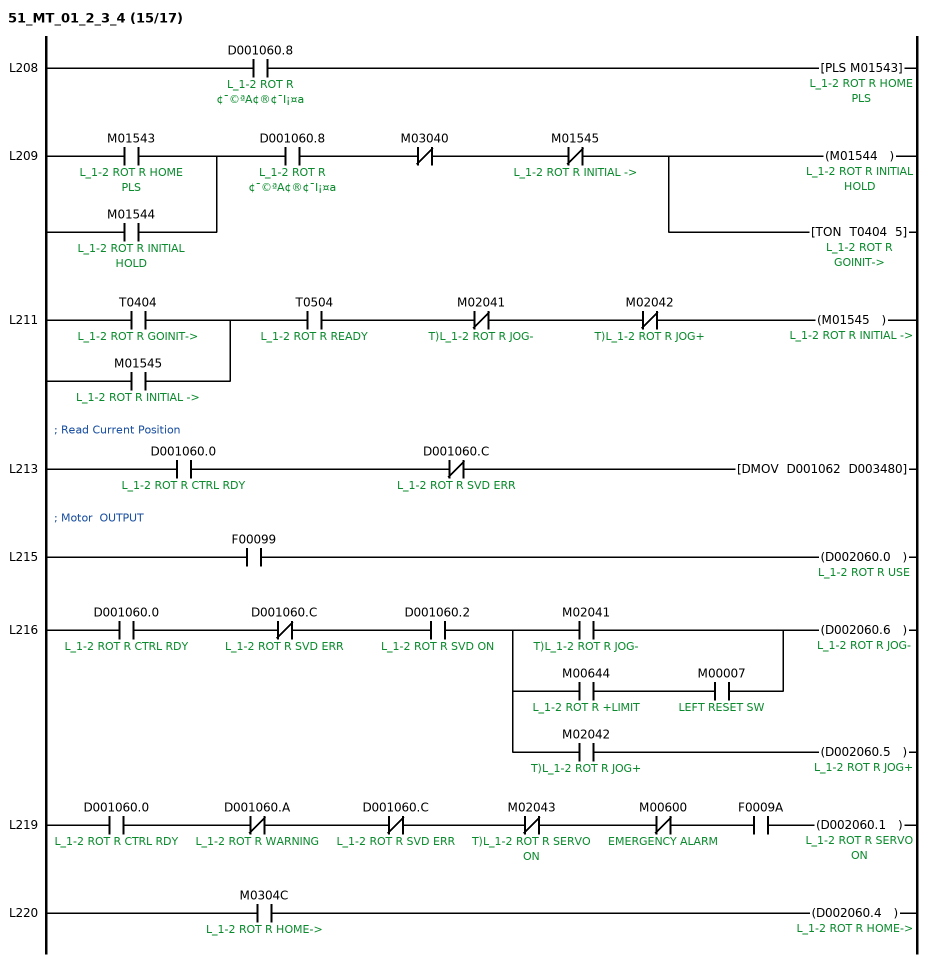
[picture p264: 51_MT_01_2_3_4 rungs L208-L220]
; L208
LOAD      D001060.8	// L_1-2 ROT R ¢¯©ªA¢®¢¯I¡¤a
OUTP      M01543	// L_1-2 ROT R HOME PLS
; L209
LOAD      M01543	// L_1-2 ROT R HOME PLS
OR        M01544	// L_1-2 ROT R INITIAL HOLD
AND       D001060.8	// L_1-2 ROT R ¢¯©ªA¢®¢¯I¡¤a
AND NOT   M03040
AND NOT   M01545	// L_1-2 ROT R INITIAL ->
OUT       M01544	// L_1-2 ROT R INITIAL HOLD
TON       T0404 5	// L_1-2 ROT R GOINIT->
; L211
LOAD      T0404	// L_1-2 ROT R GOINIT->
OR        M01545	// L_1-2 ROT R INITIAL ->
AND       T0504	// L_1-2 ROT R READY
AND NOT   M02041	// T)L_1-2 ROT R JOG-
AND NOT   M02042	// T)L_1-2 ROT R JOG+
OUT       M01545	// L_1-2 ROT R INITIAL ->
; L213
LOAD      D001060.0	// L_1-2 ROT R CTRL RDY
AND NOT   D001060.C	// L_1-2 ROT R SVD ERR
DMOV      D001062 D003480
// output comment: Read Current Position
//  Motor  OUTPUT
; L215
LOAD      F00099
OUT       D002060.0	// L_1-2 ROT R USE
; L216
LOAD      D001060.0	// L_1-2 ROT R CTRL RDY
AND NOT   D001060.C	// L_1-2 ROT R SVD ERR
AND       D001060.2	// L_1-2 ROT R SVD ON
MPUSH
LOAD      M02041	// T)L_1-2 ROT R JOG-
LOAD      M00644	// L_1-2 ROT R +LIMIT
AND       M00007	// LEFT RESET SW
OR LOAD
AND LOAD
OUT       D002060.6	// L_1-2 ROT R JOG-
MPOP
AND       M02042	// T)L_1-2 ROT R JOG+
OUT       D002060.5	// L_1-2 ROT R JOG+
; L219
LOAD      D001060.0	// L_1-2 ROT R CTRL RDY
AND NOT   D001060.A	// L_1-2 ROT R WARNING
AND NOT   D001060.C	// L_1-2 ROT R SVD ERR
AND NOT   M02043	// T)L_1-2 ROT R SERVO ON
AND NOT   M00600	// EMERGENCY ALARM
AND       F0009A
OUT       D002060.1	// L_1-2 ROT R SERVO ON
; L220
LOAD      M0304C	// L_1-2 ROT R HOME->
OUT       D002060.4	// L_1-2 ROT R HOME->

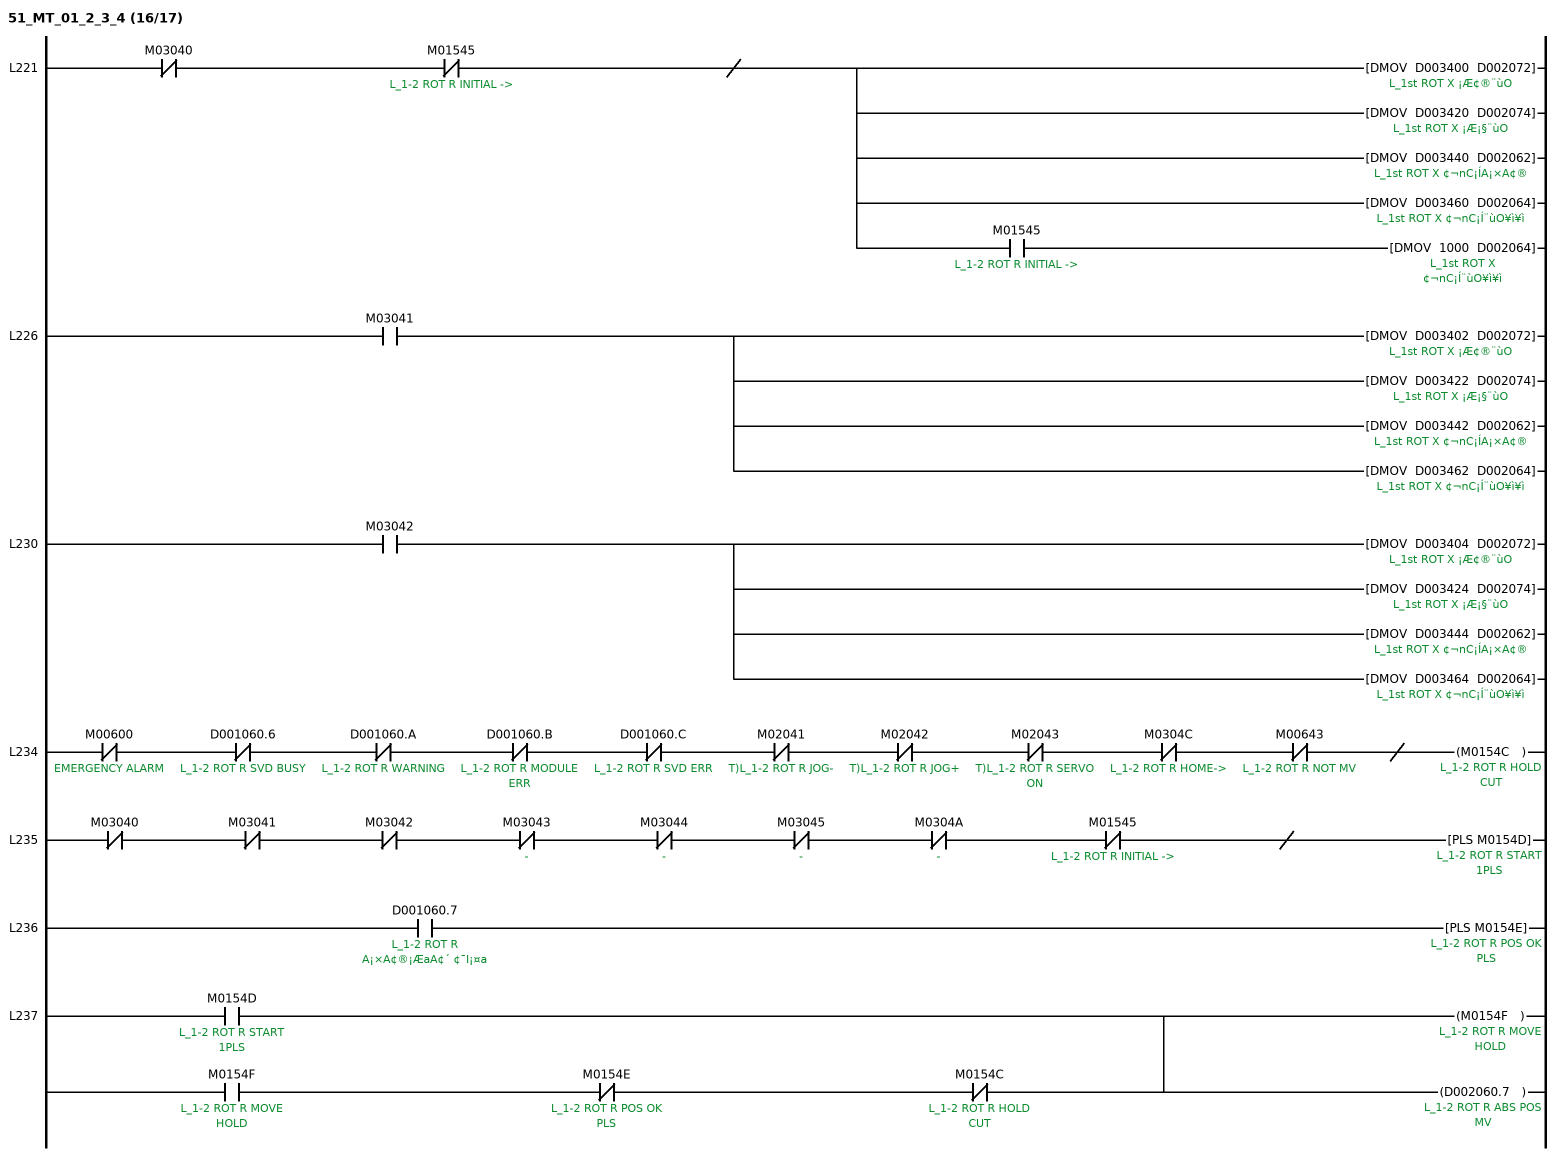
; L221
LOAD NOT  M03040
AND NOT   M01545	// L_1-2 ROT R INITIAL ->
NOT
DMOV      D003400 D002072	// L_1st ROT X ¡Æ¢®¨ùO
DMOV      D003420 D002074	// L_1st ROT X ¡Æ¡§¨ùO
DMOV      D003440 D002062	// L_1st ROT X ¢¬nC¡ÍA¡×A¢®
DMOV      D003460 D002064	// L_1st ROT X ¢¬nC¡Í¨ùO¥ì¥ì
AND       M01545	// L_1-2 ROT R INITIAL ->
DMOV      1000 D002064	// L_1st ROT X ¢¬nC¡Í¨ùO¥ì¥ì
; L226
LOAD      M03041
DMOV      D003402 D002072	// L_1st ROT X ¡Æ¢®¨ùO
DMOV      D003422 D002074	// L_1st ROT X ¡Æ¡§¨ùO
DMOV      D003442 D002062	// L_1st ROT X ¢¬nC¡ÍA¡×A¢®
DMOV      D003462 D002064	// L_1st ROT X ¢¬nC¡Í¨ùO¥ì¥ì
; L230
LOAD      M03042
DMOV      D003404 D002072	// L_1st ROT X ¡Æ¢®¨ùO
DMOV      D003424 D002074	// L_1st ROT X ¡Æ¡§¨ùO
DMOV      D003444 D002062	// L_1st ROT X ¢¬nC¡ÍA¡×A¢®
DMOV      D003464 D002064	// L_1st ROT X ¢¬nC¡Í¨ùO¥ì¥ì
; L234
LOAD NOT  M00600	// EMERGENCY ALARM
AND NOT   D001060.6	// L_1-2 ROT R SVD BUSY
AND NOT   D001060.A	// L_1-2 ROT R WARNING
AND NOT   D001060.B	// L_1-2 ROT R MODULE ERR
AND NOT   D001060.C	// L_1-2 ROT R SVD ERR
AND NOT   M02041	// T)L_1-2 ROT R JOG-
AND NOT   M02042	// T)L_1-2 ROT R JOG+
AND NOT   M02043	// T)L_1-2 ROT R SERVO ON
AND NOT   M0304C	// L_1-2 ROT R HOME->
AND NOT   M00643	// L_1-2 ROT R NOT MV
NOT
OUT       M0154C	// L_1-2 ROT R HOLD CUT
; L235
LOAD NOT  M03040
AND NOT   M03041
AND NOT   M03042
AND NOT   M03043	// -
AND NOT   M03044	// -
AND NOT   M03045	// -
AND NOT   M0304A	// -
AND NOT   M01545	// L_1-2 ROT R INITIAL ->
NOT
OUTP      M0154D	// L_1-2 ROT R START 1PLS
; L236
LOAD      D001060.7	// L_1-2 ROT R A¡×A¢®¡ÆaA¢´ ¢¯I¡¤a
OUTP      M0154E	// L_1-2 ROT R POS OK PLS
; L237
LOAD      M0154D	// L_1-2 ROT R START 1PLS
LOAD      M0154F	// L_1-2 ROT R MOVE HOLD
AND NOT   M0154E	// L_1-2 ROT R POS OK PLS
AND NOT   M0154C	// L_1-2 ROT R HOLD CUT
OR LOAD
OUT       M0154F	// L_1-2 ROT R MOVE HOLD
OUT       D002060.7	// L_1-2 ROT R ABS POS MV

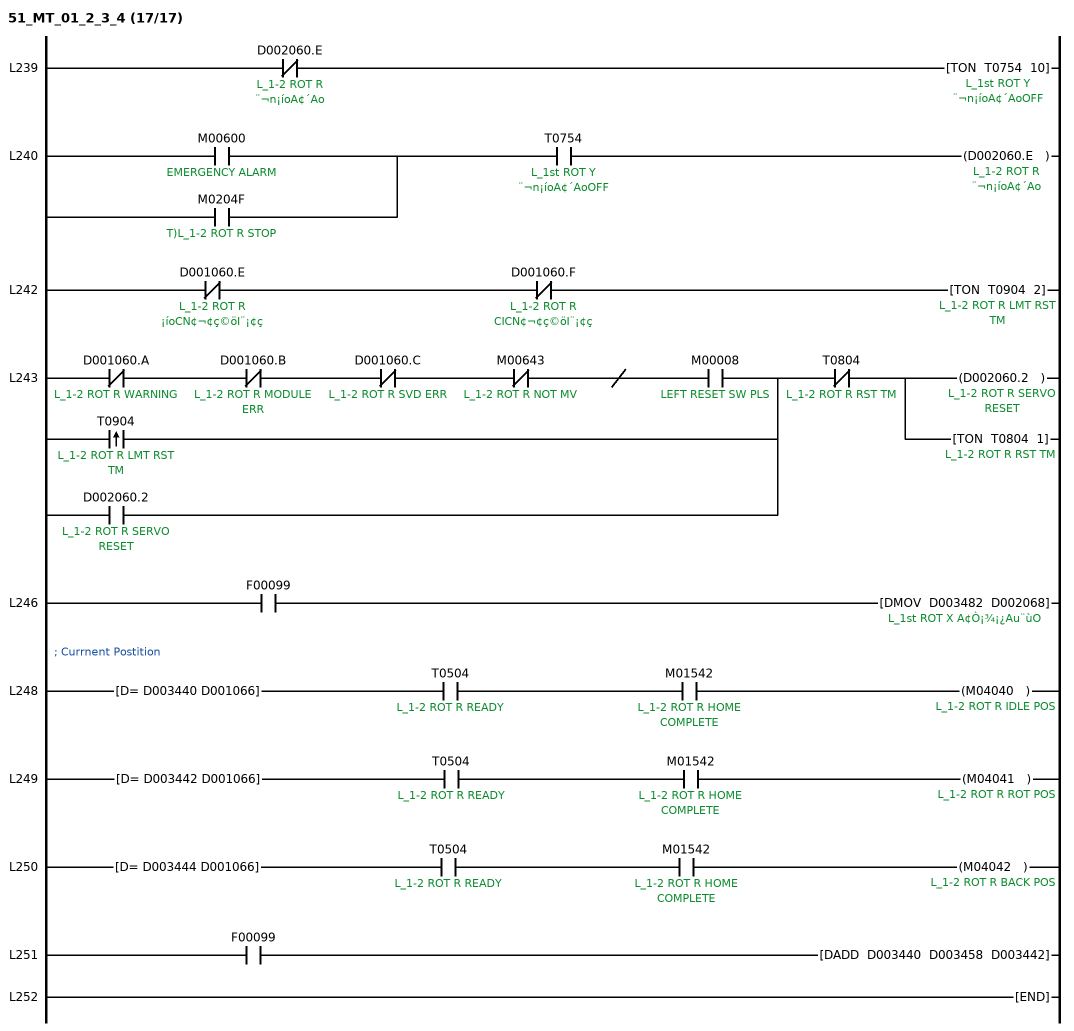
; L239
LOAD NOT  D002060.E	// L_1-2 ROT R ¨¬n¡íoA¢´Ao
TON       T0754 10	// L_1st ROT Y ¨¬n¡íoA¢´AoOFF
; L240
LOAD      M00600	// EMERGENCY ALARM
OR        M0204F	// T)L_1-2 ROT R STOP
AND       T0754	// L_1st ROT Y ¨¬n¡íoA¢´AoOFF
OUT       D002060.E	// L_1-2 ROT R ¨¬n¡íoA¢´Ao
; L242
LOAD NOT  D001060.E	// L_1-2 ROT R ¡íoCN¢¬¢ç©öI¨¡¢ç
AND NOT   D001060.F	// L_1-2 ROT R CICN¢¬¢ç©öI¨¡¢ç
TON       T0904 2	// L_1-2 ROT R LMT RST TM
; L243
LOAD NOT  D001060.A	// L_1-2 ROT R WARNING
AND NOT   D001060.B	// L_1-2 ROT R MODULE ERR
AND NOT   D001060.C	// L_1-2 ROT R SVD ERR
AND NOT   M00643	// L_1-2 ROT R NOT MV
NOT
AND       M00008	// LEFT RESET SW PLS
ORP       T0904	// L_1-2 ROT R LMT RST TM
OR        D002060.2	// L_1-2 ROT R SERVO RESET
AND NOT   T0804	// L_1-2 ROT R RST TM
OUT       D002060.2	// L_1-2 ROT R SERVO RESET
TON       T0804 1	// L_1-2 ROT R RST TM
; L246
LOAD      F00099
DMOV      D003482 D002068	// L_1st ROT X A¢Ò¡¾¡¿Au¨ùO
// Currnent Postition
; L248
LOADD=    D003440 D001066
AND       T0504	// L_1-2 ROT R READY
AND       M01542	// L_1-2 ROT R HOME COMPLETE
OUT       M04040	// L_1-2 ROT R IDLE POS
; L249
LOADD=    D003442 D001066
AND       T0504	// L_1-2 ROT R READY
AND       M01542	// L_1-2 ROT R HOME COMPLETE
OUT       M04041	// L_1-2 ROT R ROT POS
; L250
LOADD=    D003444 D001066
AND       T0504	// L_1-2 ROT R READY
AND       M01542	// L_1-2 ROT R HOME COMPLETE
OUT       M04042	// L_1-2 ROT R BACK POS
; L251
LOAD      F00099
DADD      D003440 D003458 D003442
; L252
END

PROGRAM 52_MT_05_6_7_8 (task: ¨ö¨¬A¥ì CA¡¤I¡¾¡¿¡¤¡Í)

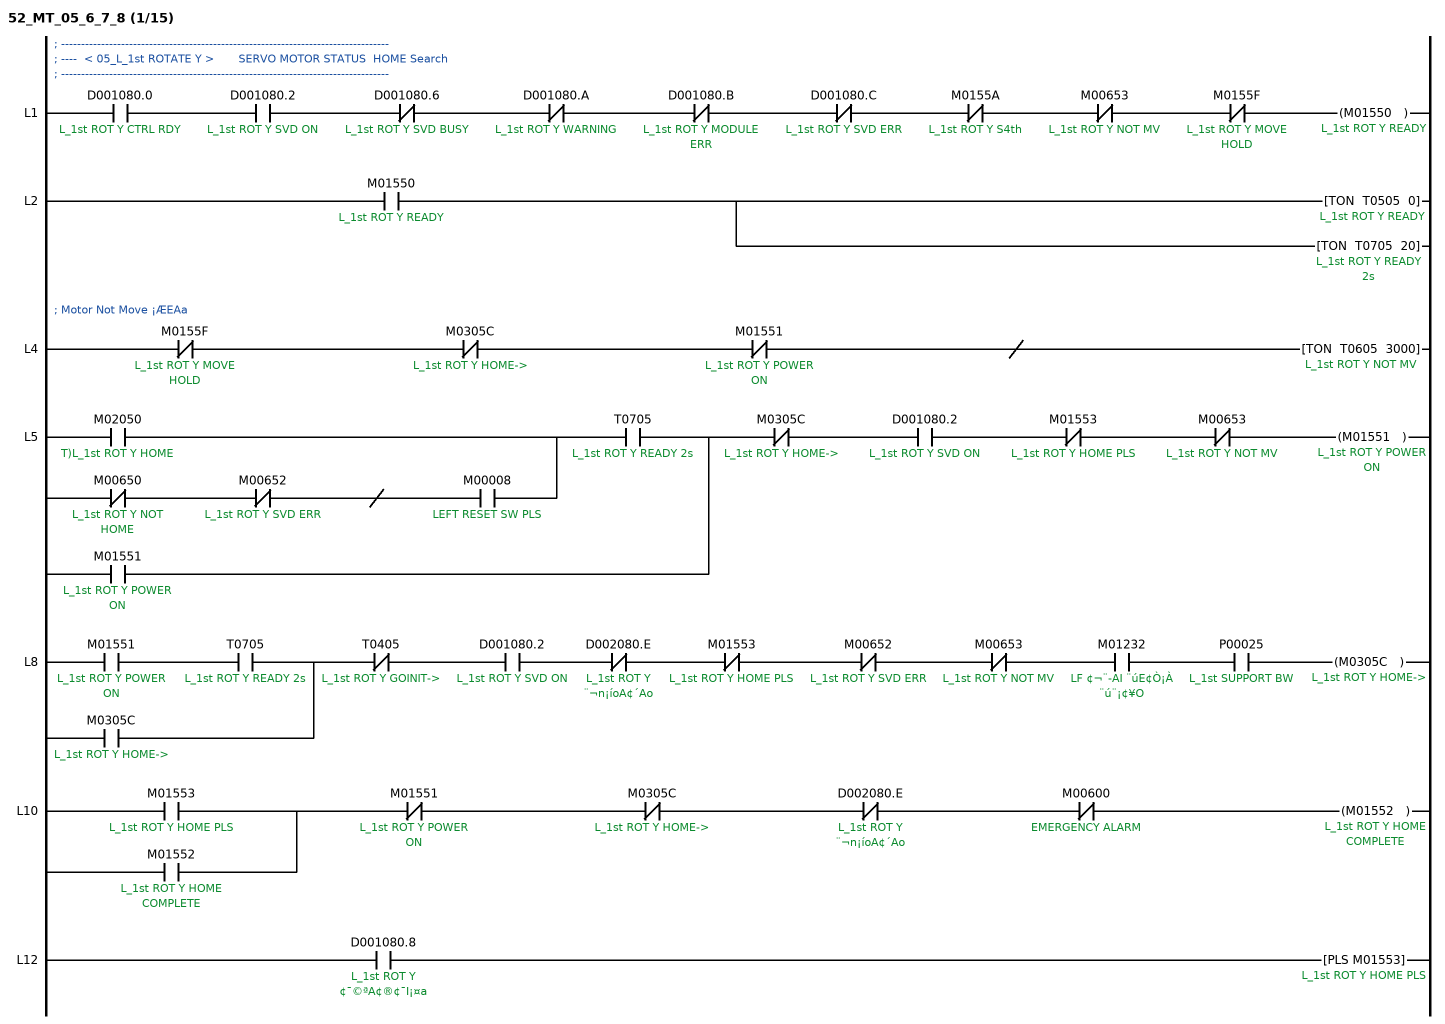
// ----------------------------------------------------------------------------------
// 
// ----  < 05_L_1st ROTATE Y >       SERVO MOTOR STATUS  HOME Search
// 
// ----------------------------------------------------------------------------------
; L1
LOAD      D001080.0	// L_1st ROT Y CTRL RDY
AND       D001080.2	// L_1st ROT Y SVD ON
AND NOT   D001080.6	// L_1st ROT Y SVD BUSY
AND NOT   D001080.A	// L_1st ROT Y WARNING
AND NOT   D001080.B	// L_1st ROT Y MODULE ERR
AND NOT   D001080.C	// L_1st ROT Y SVD ERR
AND NOT   M0155A	// L_1st ROT Y S4th
AND NOT   M00653	// L_1st ROT Y NOT MV
AND NOT   M0155F	// L_1st ROT Y MOVE HOLD
OUT       M01550	// L_1st ROT Y READY
; L2
LOAD      M01550	// L_1st ROT Y READY
TON       T0505 0	// L_1st ROT Y READY
TON       T0705 20	// L_1st ROT Y READY 2s
; L4
LOAD NOT  M0155F	// L_1st ROT Y MOVE HOLD
AND NOT   M0305C	// L_1st ROT Y HOME->
AND NOT   M01551	// L_1st ROT Y POWER ON
NOT
TON       T0605 3000	// L_1st ROT Y NOT MV
// output comment: Motor Not Move ¡ÆEAa
; L5
LOAD      M02050	// T)L_1st ROT Y HOME
LOAD NOT  M00650	// L_1st ROT Y NOT HOME
AND NOT   M00652	// L_1st ROT Y SVD ERR
NOT
AND       M00008	// LEFT RESET SW PLS
OR LOAD
AND       T0705	// L_1st ROT Y READY 2s
OR        M01551	// L_1st ROT Y POWER ON
AND NOT   M0305C	// L_1st ROT Y HOME->
AND       D001080.2	// L_1st ROT Y SVD ON
AND NOT   M01553	// L_1st ROT Y HOME PLS
AND NOT   M00653	// L_1st ROT Y NOT MV
OUT       M01551	// L_1st ROT Y POWER ON
; L8
LOAD      M01551	// L_1st ROT Y POWER ON
AND       T0705	// L_1st ROT Y READY 2s
OR        M0305C	// L_1st ROT Y HOME->
AND NOT   T0405	// L_1st ROT Y GOINIT->
AND       D001080.2	// L_1st ROT Y SVD ON
AND NOT   D002080.E	// L_1st ROT Y ¨¬n¡íoA¢´Ao
AND NOT   M01553	// L_1st ROT Y HOME PLS
AND NOT   M00652	// L_1st ROT Y SVD ERR
AND NOT   M00653	// L_1st ROT Y NOT MV
AND       M01232	// LF ¢¬¨­AI ¨úE¢Ò¡À ¨ú¨¡¢¥O
AND       P00025	// L_1st SUPPORT BW
OUT       M0305C	// L_1st ROT Y HOME->
; L10
LOAD      M01553	// L_1st ROT Y HOME PLS
OR        M01552	// L_1st ROT Y HOME COMPLETE
AND NOT   M01551	// L_1st ROT Y POWER ON
AND NOT   M0305C	// L_1st ROT Y HOME->
AND NOT   D002080.E	// L_1st ROT Y ¨¬n¡íoA¢´Ao
AND NOT   M00600	// EMERGENCY ALARM
OUT       M01552	// L_1st ROT Y HOME COMPLETE
; L12
LOAD      D001080.8	// L_1st ROT Y ¢¯©ªA¢®¢¯I¡¤a
OUTP      M01553	// L_1st ROT Y HOME PLS

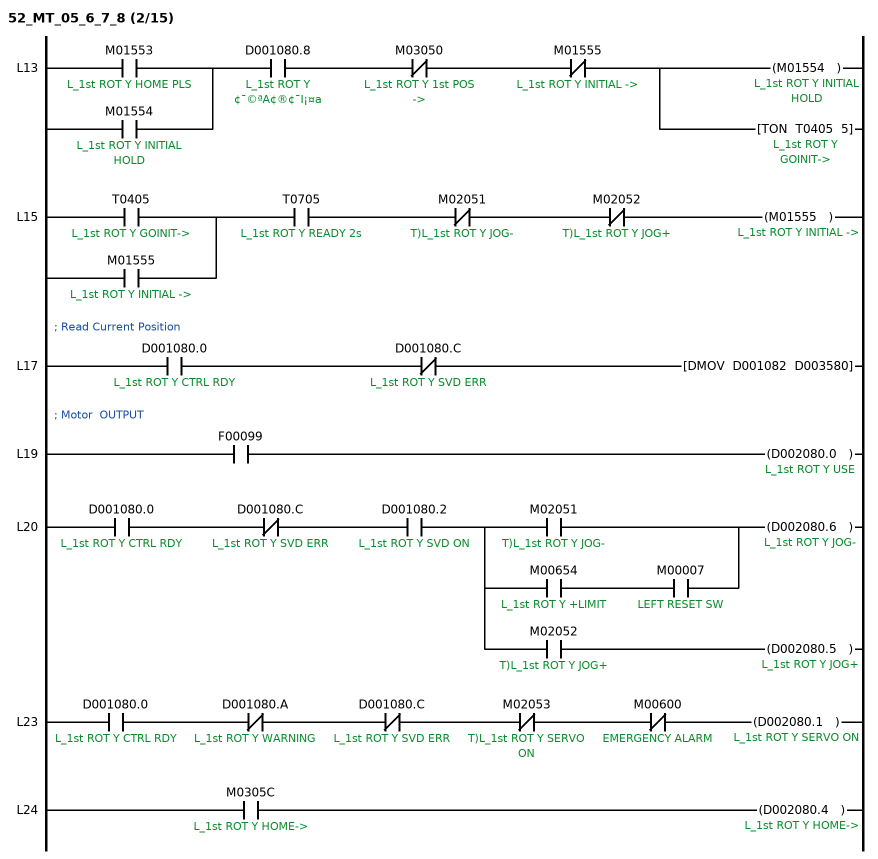
; L13
LOAD      M01553	// L_1st ROT Y HOME PLS
OR        M01554	// L_1st ROT Y INITIAL HOLD
AND       D001080.8	// L_1st ROT Y ¢¯©ªA¢®¢¯I¡¤a
AND NOT   M03050	// L_1st ROT Y 1st POS ->
AND NOT   M01555	// L_1st ROT Y INITIAL ->
OUT       M01554	// L_1st ROT Y INITIAL HOLD
TON       T0405 5	// L_1st ROT Y GOINIT->
; L15
LOAD      T0405	// L_1st ROT Y GOINIT->
OR        M01555	// L_1st ROT Y INITIAL ->
AND       T0705	// L_1st ROT Y READY 2s
AND NOT   M02051	// T)L_1st ROT Y JOG-
AND NOT   M02052	// T)L_1st ROT Y JOG+
OUT       M01555	// L_1st ROT Y INITIAL ->
; L17
LOAD      D001080.0	// L_1st ROT Y CTRL RDY
AND NOT   D001080.C	// L_1st ROT Y SVD ERR
DMOV      D001082 D003580
// output comment: Read Current Position
//  Motor  OUTPUT
; L19
LOAD      F00099
OUT       D002080.0	// L_1st ROT Y USE
; L20
LOAD      D001080.0	// L_1st ROT Y CTRL RDY
AND NOT   D001080.C	// L_1st ROT Y SVD ERR
AND       D001080.2	// L_1st ROT Y SVD ON
MPUSH
LOAD      M02051	// T)L_1st ROT Y JOG-
LOAD      M00654	// L_1st ROT Y +LIMIT
AND       M00007	// LEFT RESET SW
OR LOAD
AND LOAD
OUT       D002080.6	// L_1st ROT Y JOG-
MPOP
AND       M02052	// T)L_1st ROT Y JOG+
OUT       D002080.5	// L_1st ROT Y JOG+
; L23
LOAD      D001080.0	// L_1st ROT Y CTRL RDY
AND NOT   D001080.A	// L_1st ROT Y WARNING
AND NOT   D001080.C	// L_1st ROT Y SVD ERR
AND NOT   M02053	// T)L_1st ROT Y SERVO ON
AND NOT   M00600	// EMERGENCY ALARM
OUT       D002080.1	// L_1st ROT Y SERVO ON
; L24
LOAD      M0305C	// L_1st ROT Y HOME->
OUT       D002080.4	// L_1st ROT Y HOME->

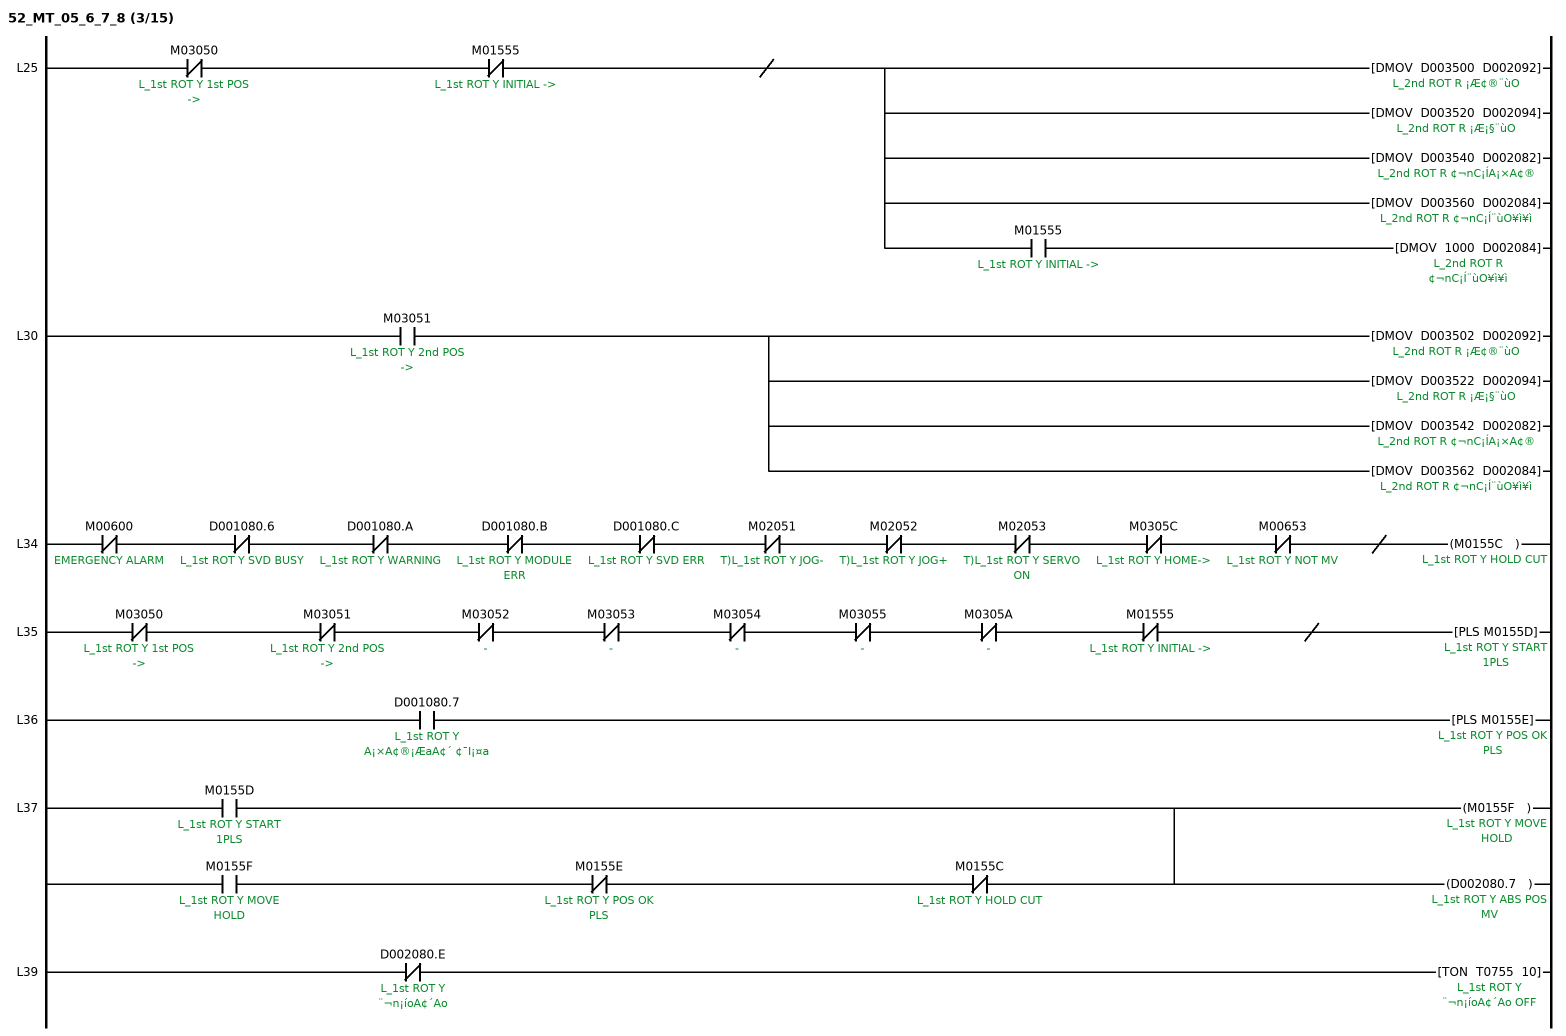
; L25
LOAD NOT  M03050	// L_1st ROT Y 1st POS ->
AND NOT   M01555	// L_1st ROT Y INITIAL ->
NOT
DMOV      D003500 D002092	// L_2nd ROT R ¡Æ¢®¨ùO
DMOV      D003520 D002094	// L_2nd ROT R ¡Æ¡§¨ùO
DMOV      D003540 D002082	// L_2nd ROT R ¢¬nC¡ÍA¡×A¢®
DMOV      D003560 D002084	// L_2nd ROT R ¢¬nC¡Í¨ùO¥ì¥ì
AND       M01555	// L_1st ROT Y INITIAL ->
DMOV      1000 D002084	// L_2nd ROT R ¢¬nC¡Í¨ùO¥ì¥ì
; L30
LOAD      M03051	// L_1st ROT Y 2nd POS ->
DMOV      D003502 D002092	// L_2nd ROT R ¡Æ¢®¨ùO
DMOV      D003522 D002094	// L_2nd ROT R ¡Æ¡§¨ùO
DMOV      D003542 D002082	// L_2nd ROT R ¢¬nC¡ÍA¡×A¢®
DMOV      D003562 D002084	// L_2nd ROT R ¢¬nC¡Í¨ùO¥ì¥ì
; L34
LOAD NOT  M00600	// EMERGENCY ALARM
AND NOT   D001080.6	// L_1st ROT Y SVD BUSY
AND NOT   D001080.A	// L_1st ROT Y WARNING
AND NOT   D001080.B	// L_1st ROT Y MODULE ERR
AND NOT   D001080.C	// L_1st ROT Y SVD ERR
AND NOT   M02051	// T)L_1st ROT Y JOG-
AND NOT   M02052	// T)L_1st ROT Y JOG+
AND NOT   M02053	// T)L_1st ROT Y SERVO ON
AND NOT   M0305C	// L_1st ROT Y HOME->
AND NOT   M00653	// L_1st ROT Y NOT MV
NOT
OUT       M0155C	// L_1st ROT Y HOLD CUT
; L35
LOAD NOT  M03050	// L_1st ROT Y 1st POS ->
AND NOT   M03051	// L_1st ROT Y 2nd POS ->
AND NOT   M03052	// -
AND NOT   M03053	// -
AND NOT   M03054	// -
AND NOT   M03055	// -
AND NOT   M0305A	// -
AND NOT   M01555	// L_1st ROT Y INITIAL ->
NOT
OUTP      M0155D	// L_1st ROT Y START 1PLS
; L36
LOAD      D001080.7	// L_1st ROT Y A¡×A¢®¡ÆaA¢´ ¢¯I¡¤a
OUTP      M0155E	// L_1st ROT Y POS OK PLS
; L37
LOAD      M0155D	// L_1st ROT Y START 1PLS
LOAD      M0155F	// L_1st ROT Y MOVE HOLD
AND NOT   M0155E	// L_1st ROT Y POS OK PLS
AND NOT   M0155C	// L_1st ROT Y HOLD CUT
OR LOAD
OUT       M0155F	// L_1st ROT Y MOVE HOLD
OUT       D002080.7	// L_1st ROT Y ABS POS MV
; L39
LOAD NOT  D002080.E	// L_1st ROT Y ¨¬n¡íoA¢´Ao
TON       T0755 10	// L_1st ROT Y ¨¬n¡íoA¢´Ao OFF

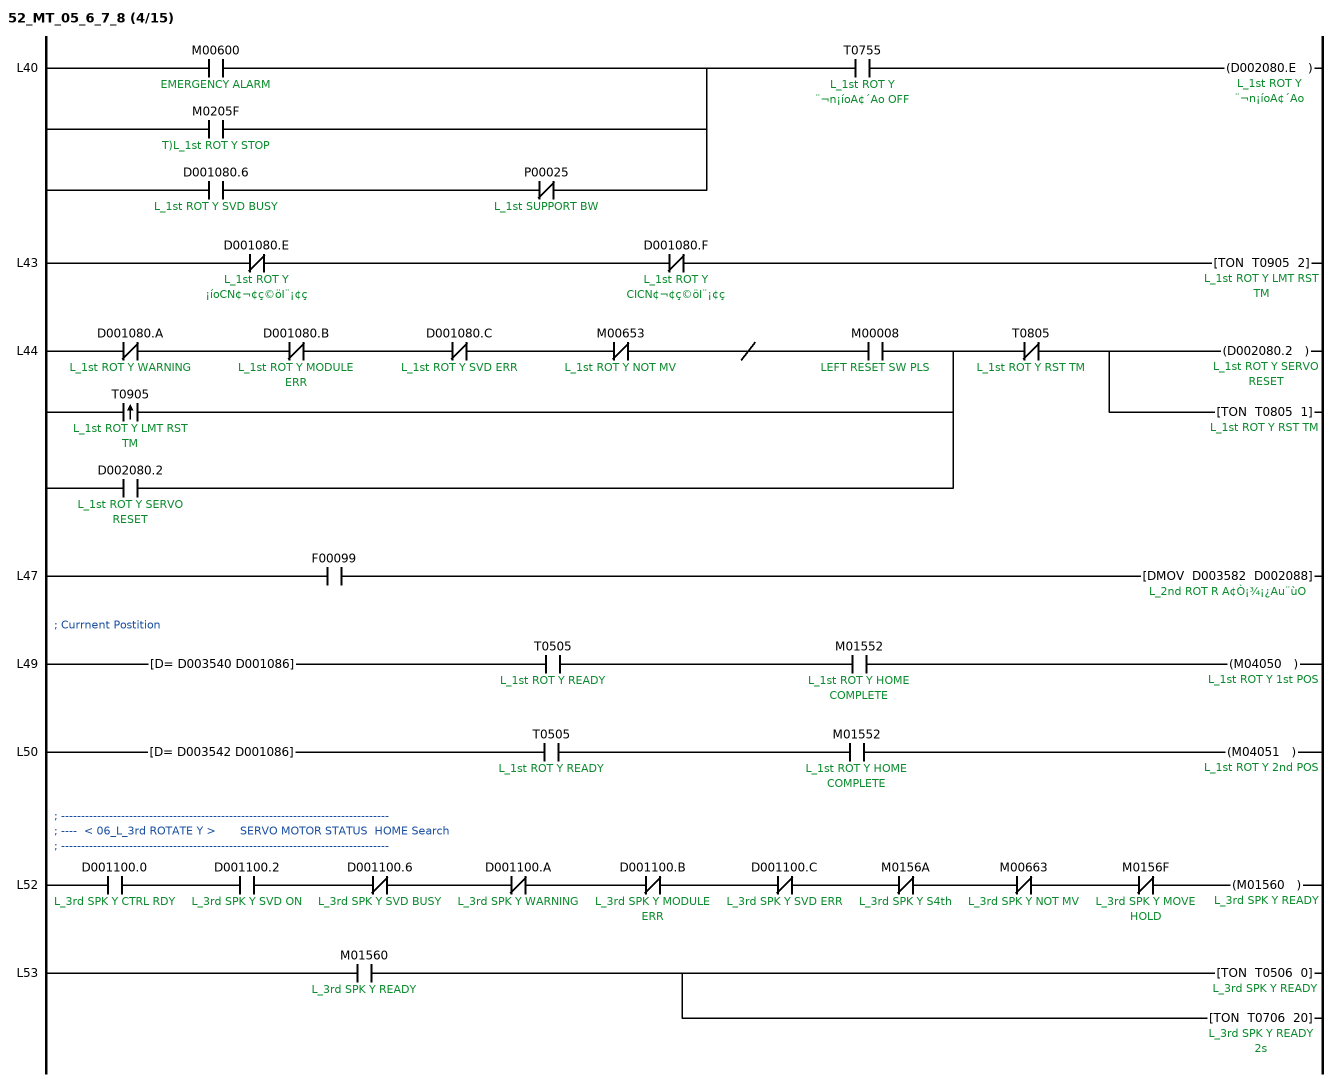
; L40
LOAD      M00600	// EMERGENCY ALARM
OR        M0205F	// T)L_1st ROT Y STOP
LOAD      D001080.6	// L_1st ROT Y SVD BUSY
AND NOT   P00025	// L_1st SUPPORT BW
OR LOAD
AND       T0755	// L_1st ROT Y ¨¬n¡íoA¢´Ao OFF
OUT       D002080.E	// L_1st ROT Y ¨¬n¡íoA¢´Ao
; L43
LOAD NOT  D001080.E	// L_1st ROT Y ¡íoCN¢¬¢ç©öI¨¡¢ç
AND NOT   D001080.F	// L_1st ROT Y CICN¢¬¢ç©öI¨¡¢ç
TON       T0905 2	// L_1st ROT Y LMT RST TM
; L44
LOAD NOT  D001080.A	// L_1st ROT Y WARNING
AND NOT   D001080.B	// L_1st ROT Y MODULE ERR
AND NOT   D001080.C	// L_1st ROT Y SVD ERR
AND NOT   M00653	// L_1st ROT Y NOT MV
NOT
AND       M00008	// LEFT RESET SW PLS
ORP       T0905	// L_1st ROT Y LMT RST TM
OR        D002080.2	// L_1st ROT Y SERVO RESET
AND NOT   T0805	// L_1st ROT Y RST TM
OUT       D002080.2	// L_1st ROT Y SERVO RESET
TON       T0805 1	// L_1st ROT Y RST TM
; L47
LOAD      F00099
DMOV      D003582 D002088	// L_2nd ROT R A¢Ò¡¾¡¿Au¨ùO
// Currnent Postition
; L49
LOADD=    D003540 D001086
AND       T0505	// L_1st ROT Y READY
AND       M01552	// L_1st ROT Y HOME COMPLETE
OUT       M04050	// L_1st ROT Y 1st POS
; L50
LOADD=    D003542 D001086
AND       T0505	// L_1st ROT Y READY
AND       M01552	// L_1st ROT Y HOME COMPLETE
OUT       M04051	// L_1st ROT Y 2nd POS
// ----------------------------------------------------------------------------------
// 
// ----  < 06_L_3rd ROTATE Y >       SERVO MOTOR STATUS  HOME Search
// 
// ----------------------------------------------------------------------------------
; L52
LOAD      D001100.0	// L_3rd SPK Y CTRL RDY
AND       D001100.2	// L_3rd SPK Y SVD ON
AND NOT   D001100.6	// L_3rd SPK Y SVD BUSY
AND NOT   D001100.A	// L_3rd SPK Y WARNING
AND NOT   D001100.B	// L_3rd SPK Y MODULE ERR
AND NOT   D001100.C	// L_3rd SPK Y SVD ERR
AND NOT   M0156A	// L_3rd SPK Y S4th
AND NOT   M00663	// L_3rd SPK Y NOT MV
AND NOT   M0156F	// L_3rd SPK Y MOVE HOLD
OUT       M01560	// L_3rd SPK Y READY
; L53
LOAD      M01560	// L_3rd SPK Y READY
TON       T0506 0	// L_3rd SPK Y READY
TON       T0706 20	// L_3rd SPK Y READY 2s

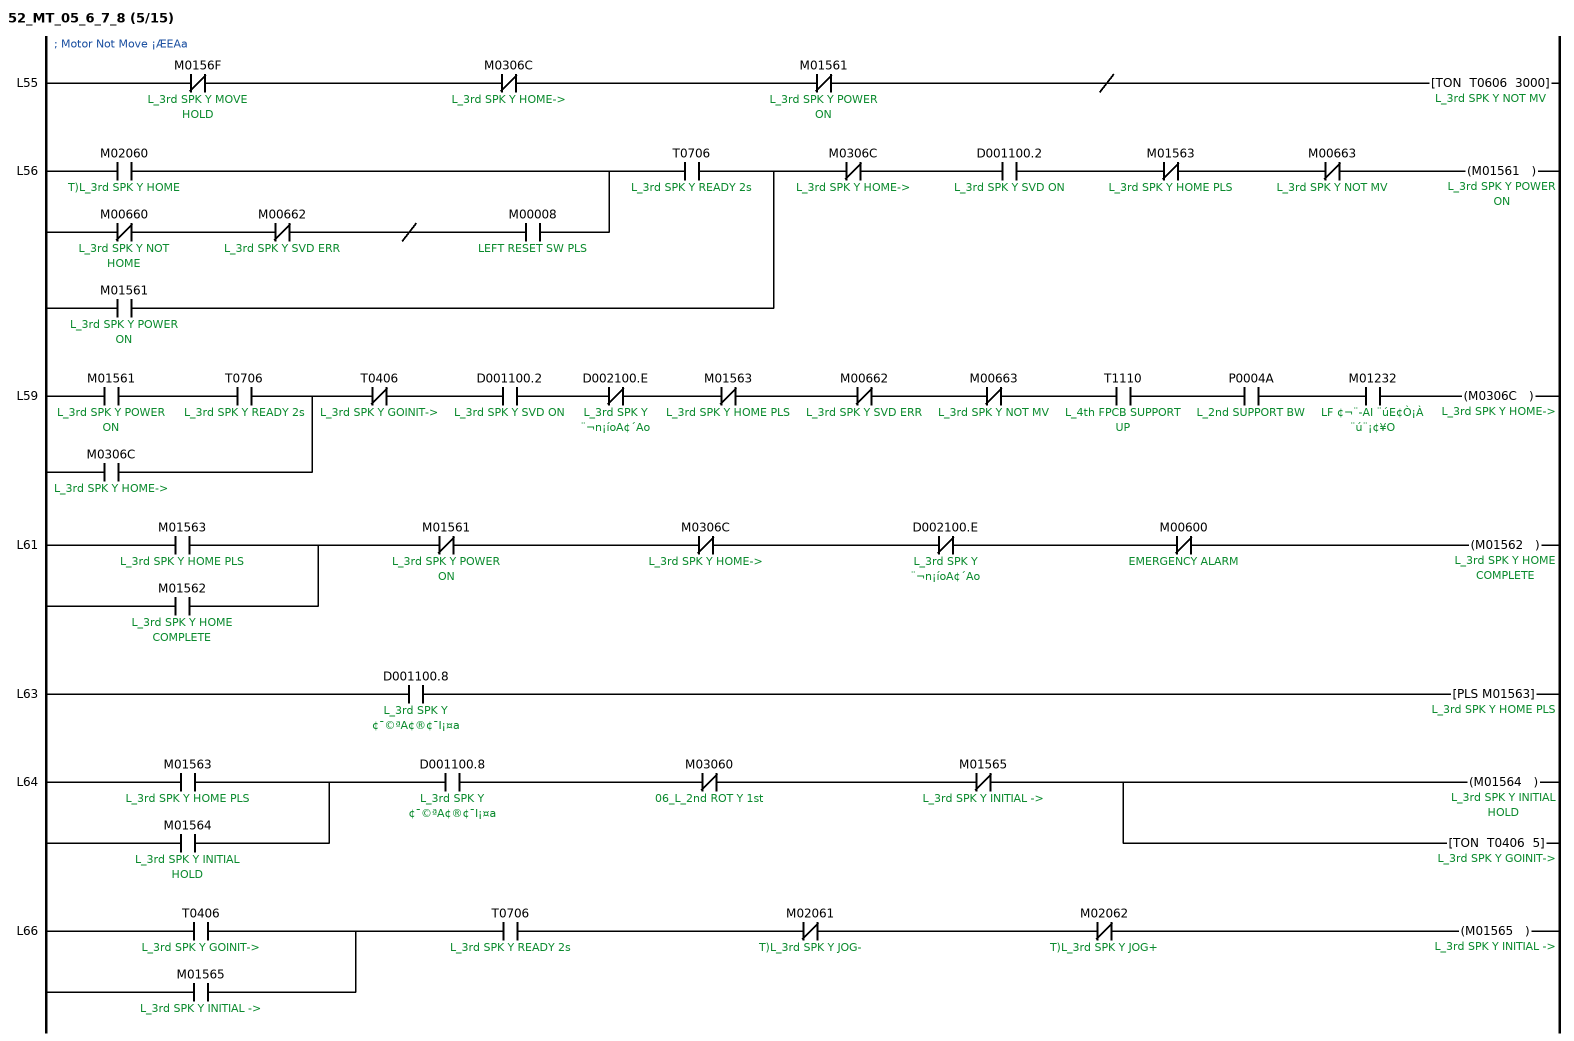
; L55
LOAD NOT  M0156F	// L_3rd SPK Y MOVE HOLD
AND NOT   M0306C	// L_3rd SPK Y HOME->
AND NOT   M01561	// L_3rd SPK Y POWER ON
NOT
TON       T0606 3000	// L_3rd SPK Y NOT MV
// output comment: Motor Not Move ¡ÆEAa
; L56
LOAD      M02060	// T)L_3rd SPK Y HOME
LOAD NOT  M00660	// L_3rd SPK Y NOT HOME
AND NOT   M00662	// L_3rd SPK Y SVD ERR
NOT
AND       M00008	// LEFT RESET SW PLS
OR LOAD
AND       T0706	// L_3rd SPK Y READY 2s
OR        M01561	// L_3rd SPK Y POWER ON
AND NOT   M0306C	// L_3rd SPK Y HOME->
AND       D001100.2	// L_3rd SPK Y SVD ON
AND NOT   M01563	// L_3rd SPK Y HOME PLS
AND NOT   M00663	// L_3rd SPK Y NOT MV
OUT       M01561	// L_3rd SPK Y POWER ON
; L59
LOAD      M01561	// L_3rd SPK Y POWER ON
AND       T0706	// L_3rd SPK Y READY 2s
OR        M0306C	// L_3rd SPK Y HOME->
AND NOT   T0406	// L_3rd SPK Y GOINIT->
AND       D001100.2	// L_3rd SPK Y SVD ON
AND NOT   D002100.E	// L_3rd SPK Y ¨¬n¡íoA¢´Ao
AND NOT   M01563	// L_3rd SPK Y HOME PLS
AND NOT   M00662	// L_3rd SPK Y SVD ERR
AND NOT   M00663	// L_3rd SPK Y NOT MV
AND       T1110	// L_4th FPCB SUPPORT UP
AND       P0004A	// L_2nd SUPPORT BW
AND       M01232	// LF ¢¬¨­AI ¨úE¢Ò¡À ¨ú¨¡¢¥O
OUT       M0306C	// L_3rd SPK Y HOME->
; L61
LOAD      M01563	// L_3rd SPK Y HOME PLS
OR        M01562	// L_3rd SPK Y HOME COMPLETE
AND NOT   M01561	// L_3rd SPK Y POWER ON
AND NOT   M0306C	// L_3rd SPK Y HOME->
AND NOT   D002100.E	// L_3rd SPK Y ¨¬n¡íoA¢´Ao
AND NOT   M00600	// EMERGENCY ALARM
OUT       M01562	// L_3rd SPK Y HOME COMPLETE
; L63
LOAD      D001100.8	// L_3rd SPK Y ¢¯©ªA¢®¢¯I¡¤a
OUTP      M01563	// L_3rd SPK Y HOME PLS
; L64
LOAD      M01563	// L_3rd SPK Y HOME PLS
OR        M01564	// L_3rd SPK Y INITIAL HOLD
AND       D001100.8	// L_3rd SPK Y ¢¯©ªA¢®¢¯I¡¤a
AND NOT   M03060	// 06_L_2nd ROT Y 1st
AND NOT   M01565	// L_3rd SPK Y INITIAL ->
OUT       M01564	// L_3rd SPK Y INITIAL HOLD
TON       T0406 5	// L_3rd SPK Y GOINIT->
; L66
LOAD      T0406	// L_3rd SPK Y GOINIT->
OR        M01565	// L_3rd SPK Y INITIAL ->
AND       T0706	// L_3rd SPK Y READY 2s
AND NOT   M02061	// T)L_3rd SPK Y JOG-
AND NOT   M02062	// T)L_3rd SPK Y JOG+
OUT       M01565	// L_3rd SPK Y INITIAL ->

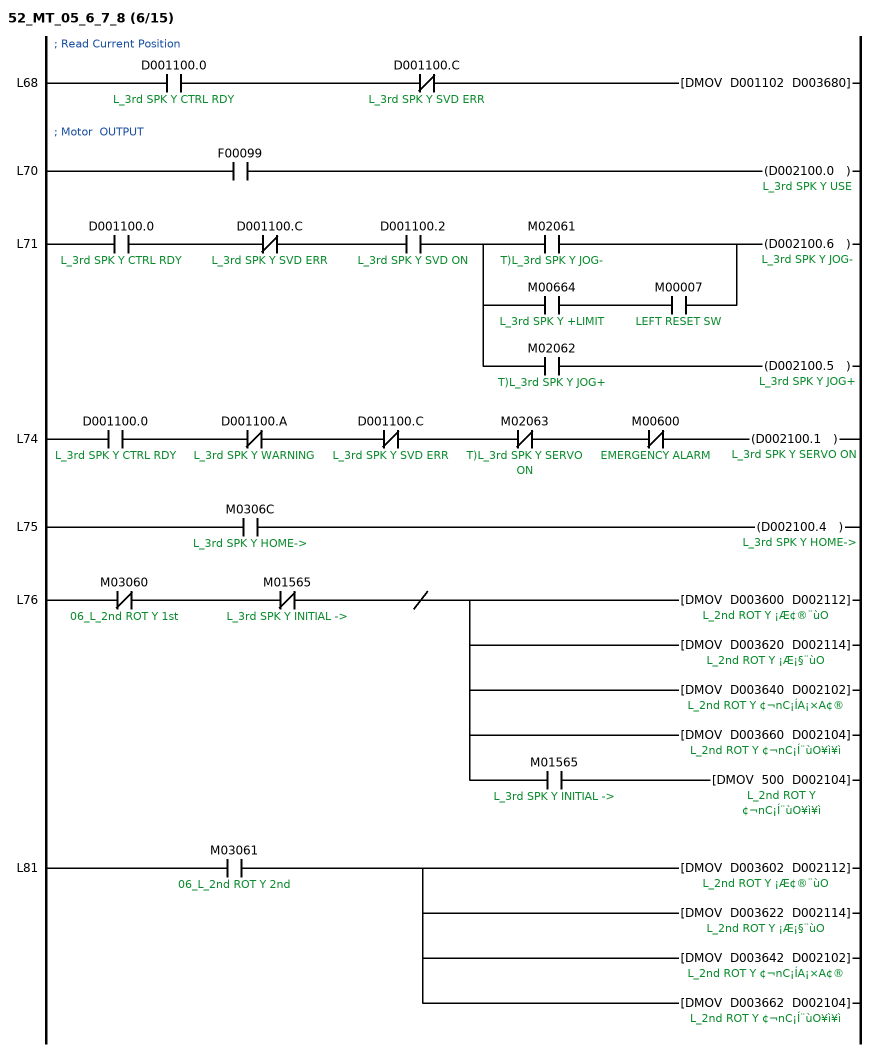
; L68
LOAD      D001100.0	// L_3rd SPK Y CTRL RDY
AND NOT   D001100.C	// L_3rd SPK Y SVD ERR
DMOV      D001102 D003680
// output comment: Read Current Position
//  Motor  OUTPUT
; L70
LOAD      F00099
OUT       D002100.0	// L_3rd SPK Y USE
; L71
LOAD      D001100.0	// L_3rd SPK Y CTRL RDY
AND NOT   D001100.C	// L_3rd SPK Y SVD ERR
AND       D001100.2	// L_3rd SPK Y SVD ON
MPUSH
LOAD      M02061	// T)L_3rd SPK Y JOG-
LOAD      M00664	// L_3rd SPK Y +LIMIT
AND       M00007	// LEFT RESET SW
OR LOAD
AND LOAD
OUT       D002100.6	// L_3rd SPK Y JOG-
MPOP
AND       M02062	// T)L_3rd SPK Y JOG+
OUT       D002100.5	// L_3rd SPK Y JOG+
; L74
LOAD      D001100.0	// L_3rd SPK Y CTRL RDY
AND NOT   D001100.A	// L_3rd SPK Y WARNING
AND NOT   D001100.C	// L_3rd SPK Y SVD ERR
AND NOT   M02063	// T)L_3rd SPK Y SERVO ON
AND NOT   M00600	// EMERGENCY ALARM
OUT       D002100.1	// L_3rd SPK Y SERVO ON
; L75
LOAD      M0306C	// L_3rd SPK Y HOME->
OUT       D002100.4	// L_3rd SPK Y HOME->
; L76
LOAD NOT  M03060	// 06_L_2nd ROT Y 1st
AND NOT   M01565	// L_3rd SPK Y INITIAL ->
NOT
DMOV      D003600 D002112	// L_2nd ROT Y ¡Æ¢®¨ùO
DMOV      D003620 D002114	// L_2nd ROT Y ¡Æ¡§¨ùO
DMOV      D003640 D002102	// L_2nd ROT Y ¢¬nC¡ÍA¡×A¢®
DMOV      D003660 D002104	// L_2nd ROT Y ¢¬nC¡Í¨ùO¥ì¥ì
AND       M01565	// L_3rd SPK Y INITIAL ->
DMOV      500 D002104	// L_2nd ROT Y ¢¬nC¡Í¨ùO¥ì¥ì
; L81
LOAD      M03061	// 06_L_2nd ROT Y 2nd
DMOV      D003602 D002112	// L_2nd ROT Y ¡Æ¢®¨ùO
DMOV      D003622 D002114	// L_2nd ROT Y ¡Æ¡§¨ùO
DMOV      D003642 D002102	// L_2nd ROT Y ¢¬nC¡ÍA¡×A¢®
DMOV      D003662 D002104	// L_2nd ROT Y ¢¬nC¡Í¨ùO¥ì¥ì

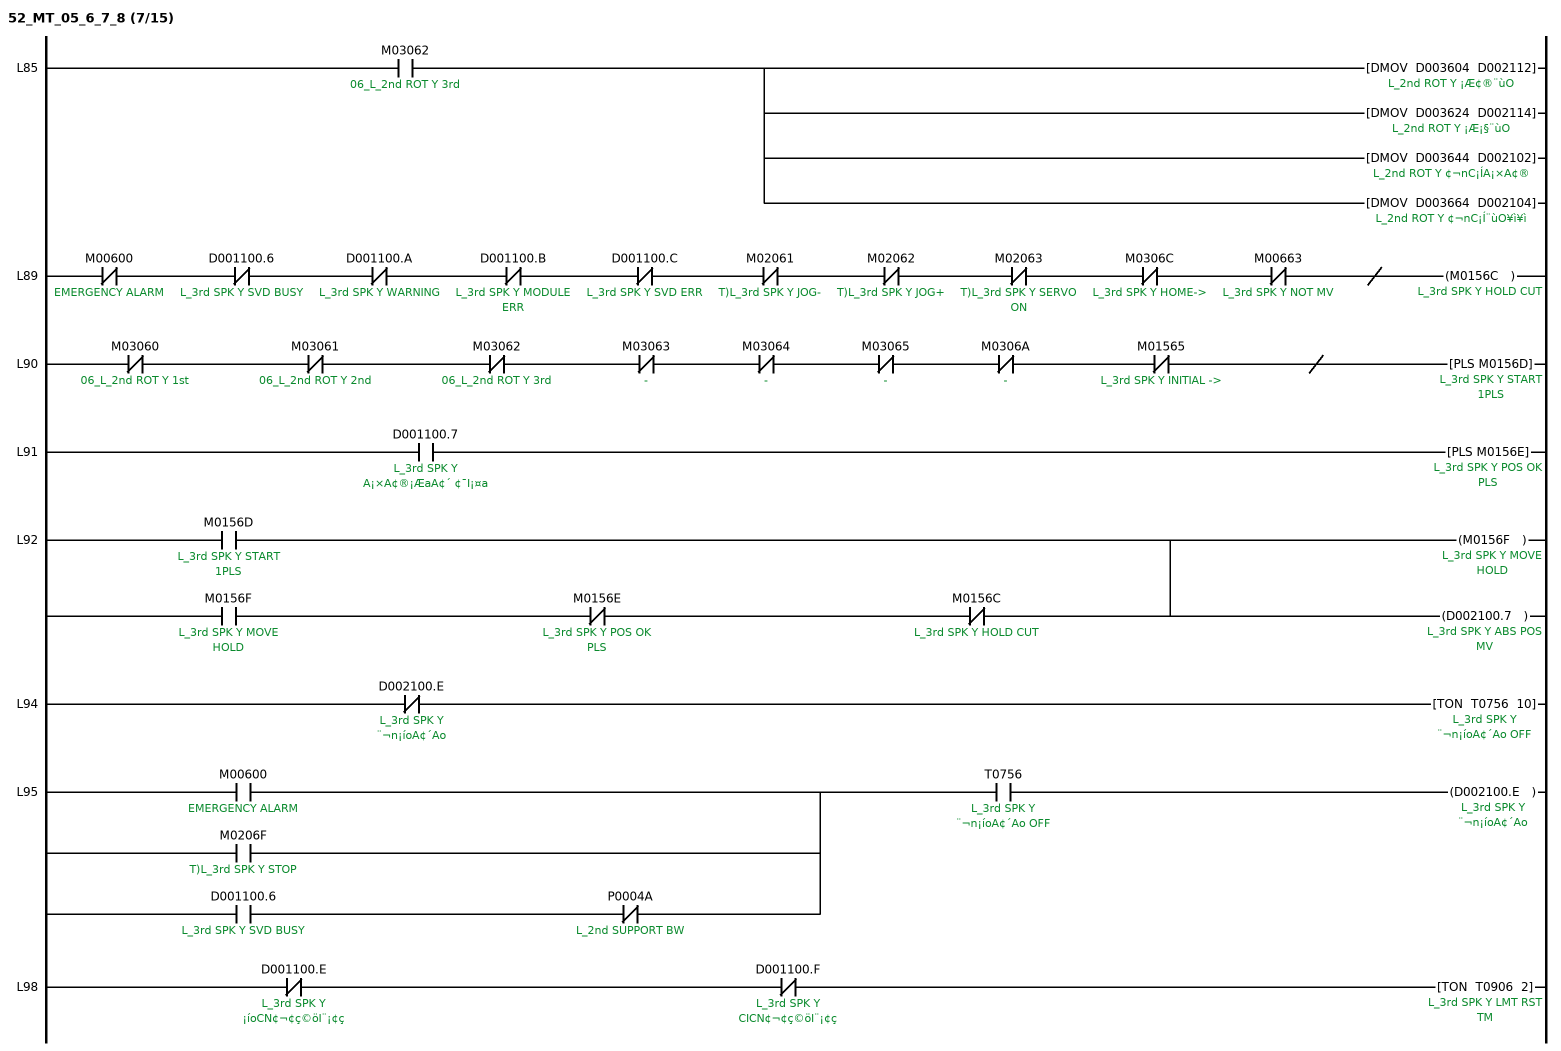
; L85
LOAD      M03062	// 06_L_2nd ROT Y 3rd
DMOV      D003604 D002112	// L_2nd ROT Y ¡Æ¢®¨ùO
DMOV      D003624 D002114	// L_2nd ROT Y ¡Æ¡§¨ùO
DMOV      D003644 D002102	// L_2nd ROT Y ¢¬nC¡ÍA¡×A¢®
DMOV      D003664 D002104	// L_2nd ROT Y ¢¬nC¡Í¨ùO¥ì¥ì
; L89
LOAD NOT  M00600	// EMERGENCY ALARM
AND NOT   D001100.6	// L_3rd SPK Y SVD BUSY
AND NOT   D001100.A	// L_3rd SPK Y WARNING
AND NOT   D001100.B	// L_3rd SPK Y MODULE ERR
AND NOT   D001100.C	// L_3rd SPK Y SVD ERR
AND NOT   M02061	// T)L_3rd SPK Y JOG-
AND NOT   M02062	// T)L_3rd SPK Y JOG+
AND NOT   M02063	// T)L_3rd SPK Y SERVO ON
AND NOT   M0306C	// L_3rd SPK Y HOME->
AND NOT   M00663	// L_3rd SPK Y NOT MV
NOT
OUT       M0156C	// L_3rd SPK Y HOLD CUT
; L90
LOAD NOT  M03060	// 06_L_2nd ROT Y 1st
AND NOT   M03061	// 06_L_2nd ROT Y 2nd
AND NOT   M03062	// 06_L_2nd ROT Y 3rd
AND NOT   M03063	// -
AND NOT   M03064	// -
AND NOT   M03065	// -
AND NOT   M0306A	// -
AND NOT   M01565	// L_3rd SPK Y INITIAL ->
NOT
OUTP      M0156D	// L_3rd SPK Y START 1PLS
; L91
LOAD      D001100.7	// L_3rd SPK Y A¡×A¢®¡ÆaA¢´ ¢¯I¡¤a
OUTP      M0156E	// L_3rd SPK Y POS OK PLS
; L92
LOAD      M0156D	// L_3rd SPK Y START 1PLS
LOAD      M0156F	// L_3rd SPK Y MOVE HOLD
AND NOT   M0156E	// L_3rd SPK Y POS OK PLS
AND NOT   M0156C	// L_3rd SPK Y HOLD CUT
OR LOAD
OUT       M0156F	// L_3rd SPK Y MOVE HOLD
OUT       D002100.7	// L_3rd SPK Y ABS POS MV
; L94
LOAD NOT  D002100.E	// L_3rd SPK Y ¨¬n¡íoA¢´Ao
TON       T0756 10	// L_3rd SPK Y ¨¬n¡íoA¢´Ao OFF
; L95
LOAD      M00600	// EMERGENCY ALARM
OR        M0206F	// T)L_3rd SPK Y STOP
LOAD      D001100.6	// L_3rd SPK Y SVD BUSY
AND NOT   P0004A	// L_2nd SUPPORT BW
OR LOAD
AND       T0756	// L_3rd SPK Y ¨¬n¡íoA¢´Ao OFF
OUT       D002100.E	// L_3rd SPK Y ¨¬n¡íoA¢´Ao
; L98
LOAD NOT  D001100.E	// L_3rd SPK Y ¡íoCN¢¬¢ç©öI¨¡¢ç
AND NOT   D001100.F	// L_3rd SPK Y CICN¢¬¢ç©öI¨¡¢ç
TON       T0906 2	// L_3rd SPK Y LMT RST TM

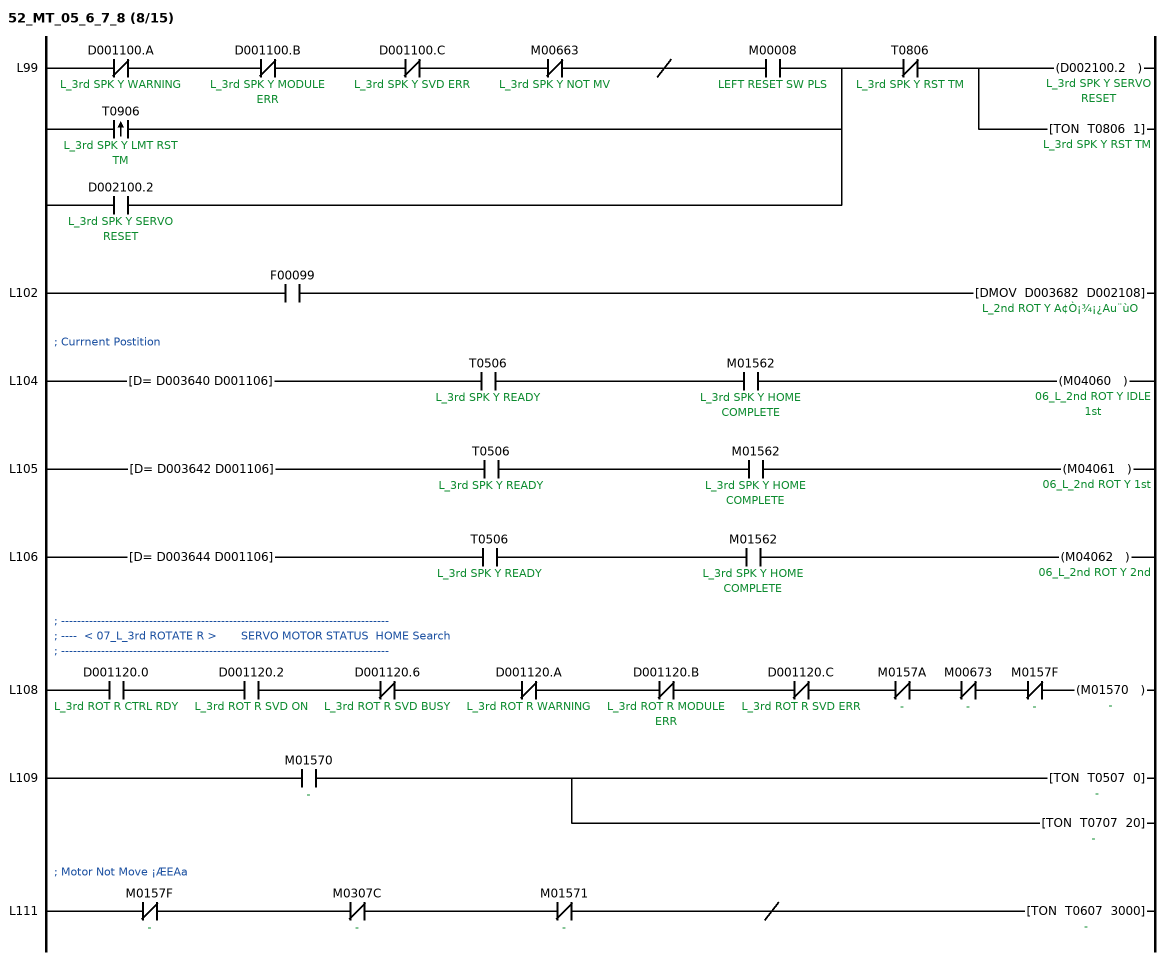
; L99
LOAD NOT  D001100.A	// L_3rd SPK Y WARNING
AND NOT   D001100.B	// L_3rd SPK Y MODULE ERR
AND NOT   D001100.C	// L_3rd SPK Y SVD ERR
AND NOT   M00663	// L_3rd SPK Y NOT MV
NOT
AND       M00008	// LEFT RESET SW PLS
ORP       T0906	// L_3rd SPK Y LMT RST TM
OR        D002100.2	// L_3rd SPK Y SERVO RESET
AND NOT   T0806	// L_3rd SPK Y RST TM
OUT       D002100.2	// L_3rd SPK Y SERVO RESET
TON       T0806 1	// L_3rd SPK Y RST TM
; L102
LOAD      F00099
DMOV      D003682 D002108	// L_2nd ROT Y A¢Ò¡¾¡¿Au¨ùO
// Currnent Postition
; L104
LOADD=    D003640 D001106
AND       T0506	// L_3rd SPK Y READY
AND       M01562	// L_3rd SPK Y HOME COMPLETE
OUT       M04060	// 06_L_2nd ROT Y IDLE 1st
; L105
LOADD=    D003642 D001106
AND       T0506	// L_3rd SPK Y READY
AND       M01562	// L_3rd SPK Y HOME COMPLETE
OUT       M04061	// 06_L_2nd ROT Y 1st
; L106
LOADD=    D003644 D001106
AND       T0506	// L_3rd SPK Y READY
AND       M01562	// L_3rd SPK Y HOME COMPLETE
OUT       M04062	// 06_L_2nd ROT Y 2nd
// ----------------------------------------------------------------------------------
// 
// ----  < 07_L_3rd ROTATE R >       SERVO MOTOR STATUS  HOME Search
// 
// ----------------------------------------------------------------------------------
; L108
LOAD      D001120.0	// L_3rd ROT R CTRL RDY
AND       D001120.2	// L_3rd ROT R SVD ON
AND NOT   D001120.6	// L_3rd ROT R SVD BUSY
AND NOT   D001120.A	// L_3rd ROT R WARNING
AND NOT   D001120.B	// L_3rd ROT R MODULE ERR
AND NOT   D001120.C	// L_3rd ROT R SVD ERR
AND NOT   M0157A	// -
AND NOT   M00673	// -
AND NOT   M0157F	// -
OUT       M01570	// -
; L109
LOAD      M01570	// -
TON       T0507 0	// -
TON       T0707 20	// -
; L111
LOAD NOT  M0157F	// -
AND NOT   M0307C	// -
AND NOT   M01571	// -
NOT
TON       T0607 3000	// -
// output comment: Motor Not Move ¡ÆEAa

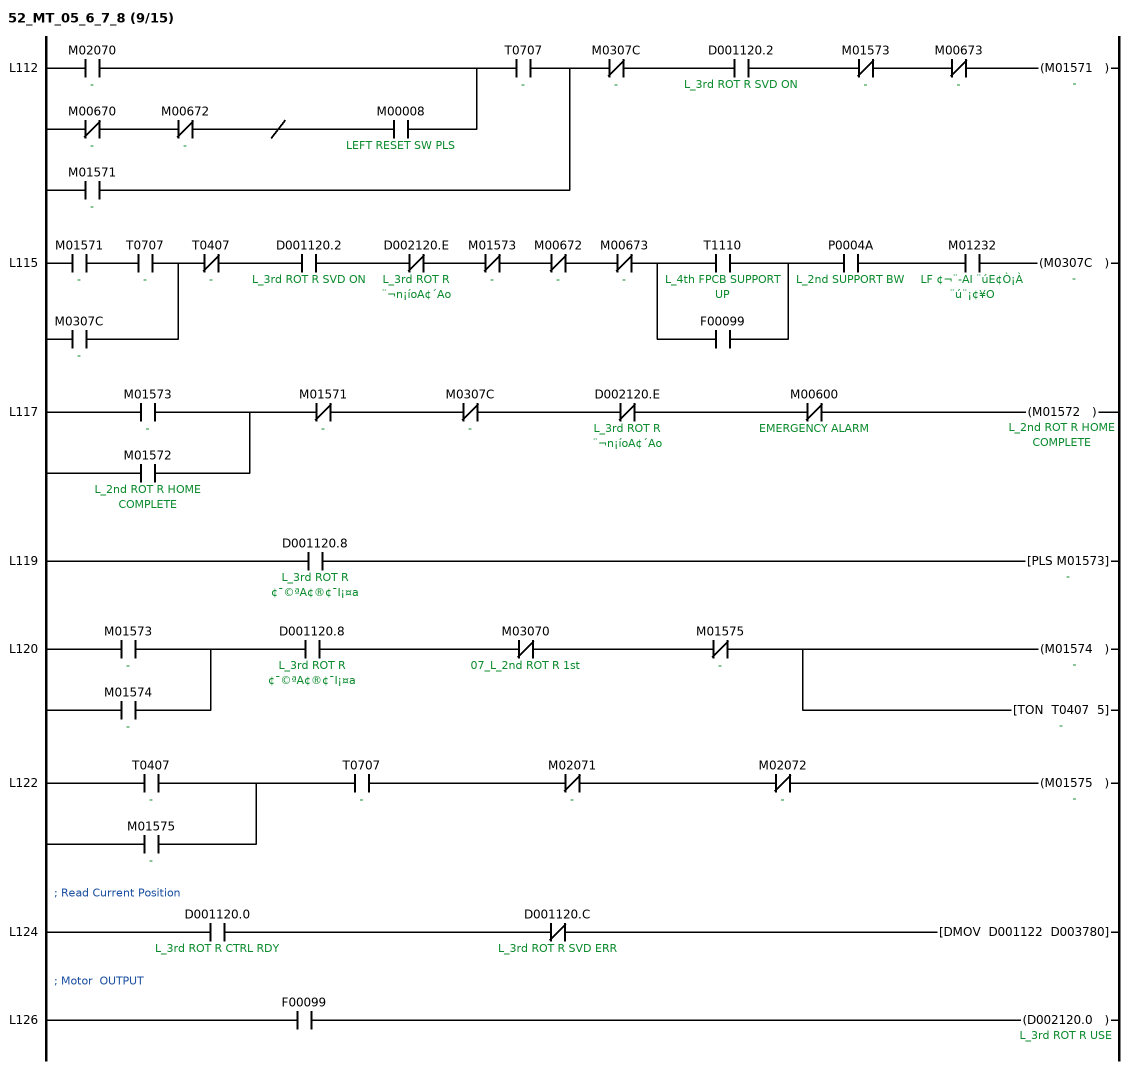
; L112
LOAD      M02070	// -
LOAD NOT  M00670	// -
AND NOT   M00672	// -
NOT
AND       M00008	// LEFT RESET SW PLS
OR LOAD
AND       T0707	// -
OR        M01571	// -
AND NOT   M0307C	// -
AND       D001120.2	// L_3rd ROT R SVD ON
AND NOT   M01573	// -
AND NOT   M00673	// -
OUT       M01571	// -
; L115
LOAD      M01571	// -
AND       T0707	// -
OR        M0307C	// -
AND NOT   T0407	// -
AND       D001120.2	// L_3rd ROT R SVD ON
AND NOT   D002120.E	// L_3rd ROT R ¨¬n¡íoA¢´Ao
AND NOT   M01573	// -
AND NOT   M00672	// -
AND NOT   M00673	// -
LOAD      T1110	// L_4th FPCB SUPPORT UP
OR        F00099
AND LOAD
AND       P0004A	// L_2nd SUPPORT BW
AND       M01232	// LF ¢¬¨­AI ¨úE¢Ò¡À ¨ú¨¡¢¥O
OUT       M0307C	// -
; L117
LOAD      M01573	// -
OR        M01572	// L_2nd ROT R HOME COMPLETE
AND NOT   M01571	// -
AND NOT   M0307C	// -
AND NOT   D002120.E	// L_3rd ROT R ¨¬n¡íoA¢´Ao
AND NOT   M00600	// EMERGENCY ALARM
OUT       M01572	// L_2nd ROT R HOME COMPLETE
; L119
LOAD      D001120.8	// L_3rd ROT R ¢¯©ªA¢®¢¯I¡¤a
OUTP      M01573	// -
; L120
LOAD      M01573	// -
OR        M01574	// -
AND       D001120.8	// L_3rd ROT R ¢¯©ªA¢®¢¯I¡¤a
AND NOT   M03070	// 07_L_2nd ROT R 1st
AND NOT   M01575	// -
OUT       M01574	// -
TON       T0407 5	// -
; L122
LOAD      T0407	// -
OR        M01575	// -
AND       T0707	// -
AND NOT   M02071	// -
AND NOT   M02072	// -
OUT       M01575	// -
; L124
LOAD      D001120.0	// L_3rd ROT R CTRL RDY
AND NOT   D001120.C	// L_3rd ROT R SVD ERR
DMOV      D001122 D003780
// output comment: Read Current Position
//  Motor  OUTPUT
; L126
LOAD      F00099
OUT       D002120.0	// L_3rd ROT R USE

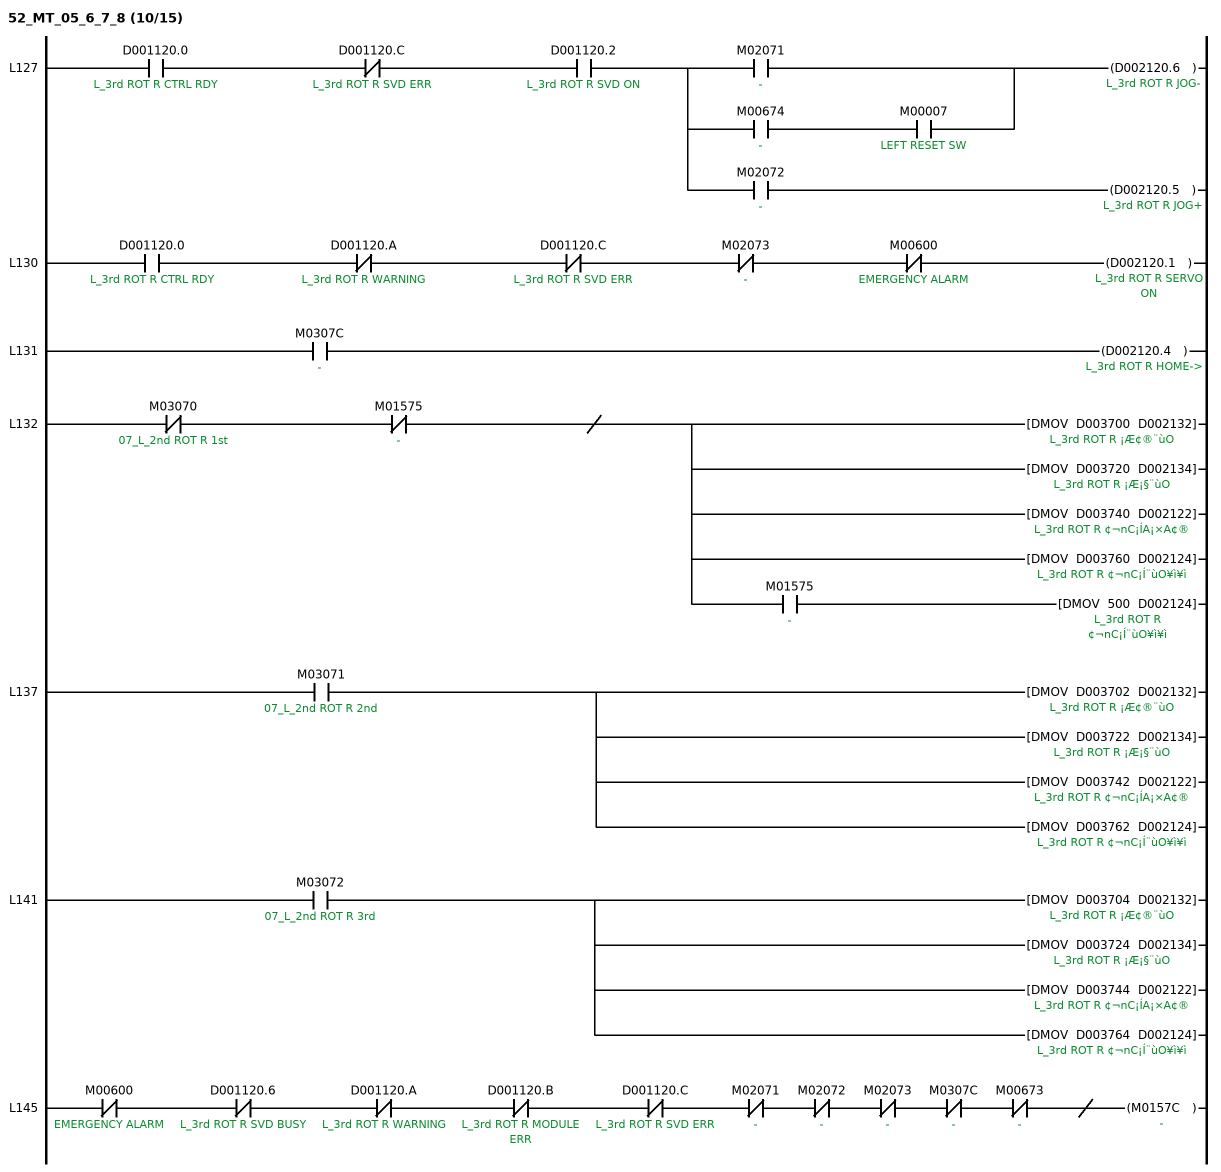
; L127
LOAD      D001120.0	// L_3rd ROT R CTRL RDY
AND NOT   D001120.C	// L_3rd ROT R SVD ERR
AND       D001120.2	// L_3rd ROT R SVD ON
MPUSH
LOAD      M02071	// -
LOAD      M00674	// -
AND       M00007	// LEFT RESET SW
OR LOAD
AND LOAD
OUT       D002120.6	// L_3rd ROT R JOG-
MPOP
AND       M02072	// -
OUT       D002120.5	// L_3rd ROT R JOG+
; L130
LOAD      D001120.0	// L_3rd ROT R CTRL RDY
AND NOT   D001120.A	// L_3rd ROT R WARNING
AND NOT   D001120.C	// L_3rd ROT R SVD ERR
AND NOT   M02073	// -
AND NOT   M00600	// EMERGENCY ALARM
OUT       D002120.1	// L_3rd ROT R SERVO ON
; L131
LOAD      M0307C	// -
OUT       D002120.4	// L_3rd ROT R HOME->
; L132
LOAD NOT  M03070	// 07_L_2nd ROT R 1st
AND NOT   M01575	// -
NOT
DMOV      D003700 D002132	// L_3rd ROT R ¡Æ¢®¨ùO
DMOV      D003720 D002134	// L_3rd ROT R ¡Æ¡§¨ùO
DMOV      D003740 D002122	// L_3rd ROT R ¢¬nC¡ÍA¡×A¢®
DMOV      D003760 D002124	// L_3rd ROT R ¢¬nC¡Í¨ùO¥ì¥ì
AND       M01575	// -
DMOV      500 D002124	// L_3rd ROT R ¢¬nC¡Í¨ùO¥ì¥ì
; L137
LOAD      M03071	// 07_L_2nd ROT R 2nd
DMOV      D003702 D002132	// L_3rd ROT R ¡Æ¢®¨ùO
DMOV      D003722 D002134	// L_3rd ROT R ¡Æ¡§¨ùO
DMOV      D003742 D002122	// L_3rd ROT R ¢¬nC¡ÍA¡×A¢®
DMOV      D003762 D002124	// L_3rd ROT R ¢¬nC¡Í¨ùO¥ì¥ì
; L141
LOAD      M03072	// 07_L_2nd ROT R 3rd
DMOV      D003704 D002132	// L_3rd ROT R ¡Æ¢®¨ùO
DMOV      D003724 D002134	// L_3rd ROT R ¡Æ¡§¨ùO
DMOV      D003744 D002122	// L_3rd ROT R ¢¬nC¡ÍA¡×A¢®
DMOV      D003764 D002124	// L_3rd ROT R ¢¬nC¡Í¨ùO¥ì¥ì
; L145
LOAD NOT  M00600	// EMERGENCY ALARM
AND NOT   D001120.6	// L_3rd ROT R SVD BUSY
AND NOT   D001120.A	// L_3rd ROT R WARNING
AND NOT   D001120.B	// L_3rd ROT R MODULE ERR
AND NOT   D001120.C	// L_3rd ROT R SVD ERR
AND NOT   M02071	// -
AND NOT   M02072	// -
AND NOT   M02073	// -
AND NOT   M0307C	// -
AND NOT   M00673	// -
NOT
OUT       M0157C	// -

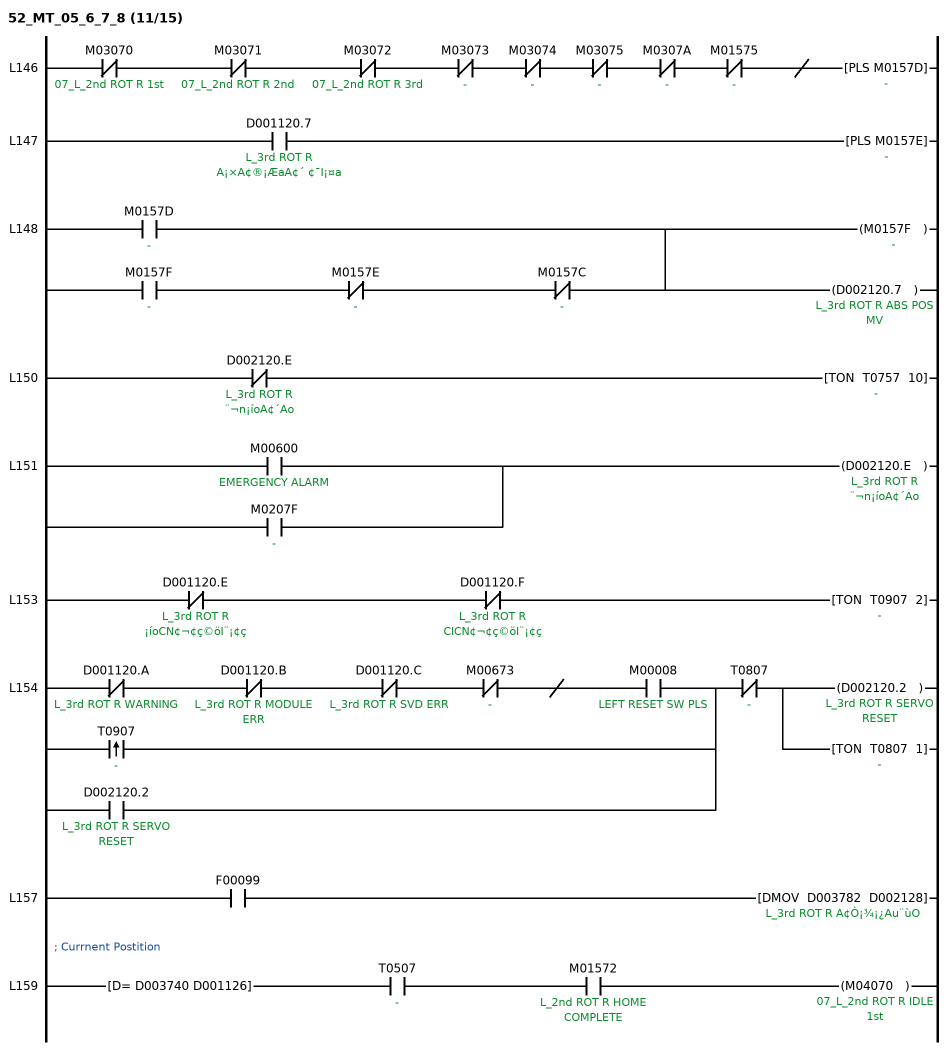
; L146
LOAD NOT  M03070	// 07_L_2nd ROT R 1st
AND NOT   M03071	// 07_L_2nd ROT R 2nd
AND NOT   M03072	// 07_L_2nd ROT R 3rd
AND NOT   M03073	// -
AND NOT   M03074	// -
AND NOT   M03075	// -
AND NOT   M0307A	// -
AND NOT   M01575	// -
NOT
OUTP      M0157D	// -
; L147
LOAD      D001120.7	// L_3rd ROT R A¡×A¢®¡ÆaA¢´ ¢¯I¡¤a
OUTP      M0157E	// -
; L148
LOAD      M0157D	// -
LOAD      M0157F	// -
AND NOT   M0157E	// -
AND NOT   M0157C	// -
OR LOAD
OUT       M0157F	// -
OUT       D002120.7	// L_3rd ROT R ABS POS MV
; L150
LOAD NOT  D002120.E	// L_3rd ROT R ¨¬n¡íoA¢´Ao
TON       T0757 10	// -
; L151
LOAD      M00600	// EMERGENCY ALARM
OR        M0207F	// -
OUT       D002120.E	// L_3rd ROT R ¨¬n¡íoA¢´Ao
; L153
LOAD NOT  D001120.E	// L_3rd ROT R ¡íoCN¢¬¢ç©öI¨¡¢ç
AND NOT   D001120.F	// L_3rd ROT R CICN¢¬¢ç©öI¨¡¢ç
TON       T0907 2	// -
; L154
LOAD NOT  D001120.A	// L_3rd ROT R WARNING
AND NOT   D001120.B	// L_3rd ROT R MODULE ERR
AND NOT   D001120.C	// L_3rd ROT R SVD ERR
AND NOT   M00673	// -
NOT
AND       M00008	// LEFT RESET SW PLS
ORP       T0907	// -
OR        D002120.2	// L_3rd ROT R SERVO RESET
AND NOT   T0807	// -
OUT       D002120.2	// L_3rd ROT R SERVO RESET
TON       T0807 1	// -
; L157
LOAD      F00099
DMOV      D003782 D002128	// L_3rd ROT R A¢Ò¡¾¡¿Au¨ùO
// Currnent Postition
; L159
LOADD=    D003740 D001126
AND       T0507	// -
AND       M01572	// L_2nd ROT R HOME COMPLETE
OUT       M04070	// 07_L_2nd ROT R IDLE 1st

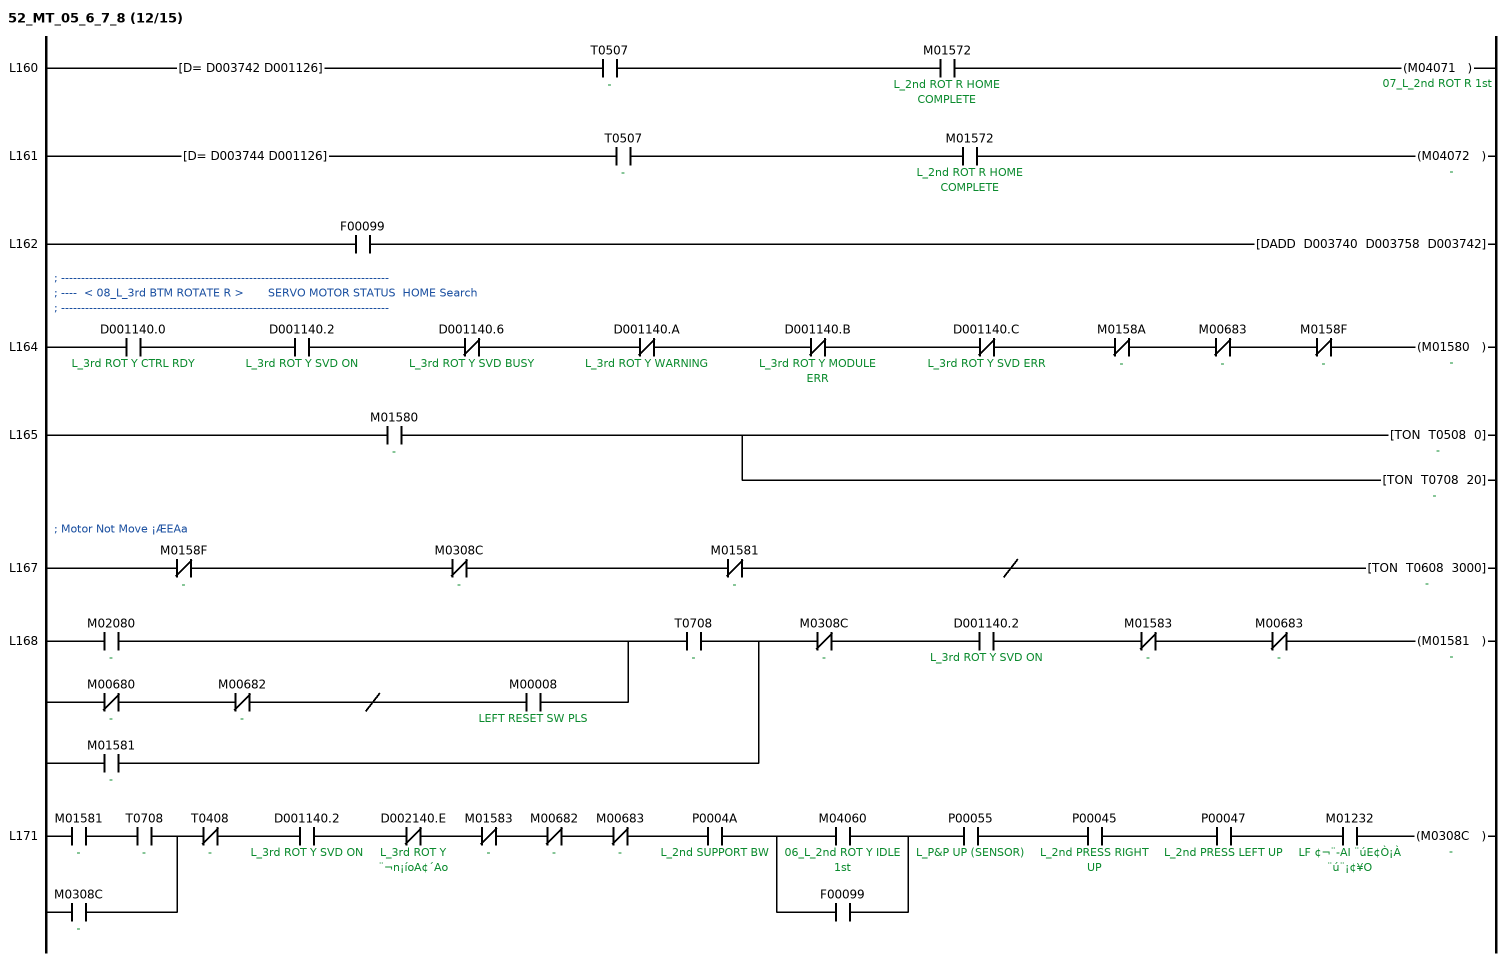
; L160
LOADD=    D003742 D001126
AND       T0507	// -
AND       M01572	// L_2nd ROT R HOME COMPLETE
OUT       M04071	// 07_L_2nd ROT R 1st
; L161
LOADD=    D003744 D001126
AND       T0507	// -
AND       M01572	// L_2nd ROT R HOME COMPLETE
OUT       M04072	// -
; L162
LOAD      F00099
DADD      D003740 D003758 D003742
// ----------------------------------------------------------------------------------
// 
// ----  < 08_L_3rd BTM ROTATE R >       SERVO MOTOR STATUS  HOME Search
// 
// ----------------------------------------------------------------------------------
; L164
LOAD      D001140.0	// L_3rd ROT Y CTRL RDY
AND       D001140.2	// L_3rd ROT Y SVD ON
AND NOT   D001140.6	// L_3rd ROT Y SVD BUSY
AND NOT   D001140.A	// L_3rd ROT Y WARNING
AND NOT   D001140.B	// L_3rd ROT Y MODULE ERR
AND NOT   D001140.C	// L_3rd ROT Y SVD ERR
AND NOT   M0158A	// -
AND NOT   M00683	// -
AND NOT   M0158F	// -
OUT       M01580	// -
; L165
LOAD      M01580	// -
TON       T0508 0	// -
TON       T0708 20	// -
; L167
LOAD NOT  M0158F	// -
AND NOT   M0308C	// -
AND NOT   M01581	// -
NOT
TON       T0608 3000	// -
// output comment: Motor Not Move ¡ÆEAa
; L168
LOAD      M02080	// -
LOAD NOT  M00680	// -
AND NOT   M00682	// -
NOT
AND       M00008	// LEFT RESET SW PLS
OR LOAD
AND       T0708	// -
OR        M01581	// -
AND NOT   M0308C	// -
AND       D001140.2	// L_3rd ROT Y SVD ON
AND NOT   M01583	// -
AND NOT   M00683	// -
OUT       M01581	// -
; L171
LOAD      M01581	// -
AND       T0708	// -
OR        M0308C	// -
AND NOT   T0408	// -
AND       D001140.2	// L_3rd ROT Y SVD ON
AND NOT   D002140.E	// L_3rd ROT Y ¨¬n¡íoA¢´Ao
AND NOT   M01583	// -
AND NOT   M00682	// -
AND NOT   M00683	// -
AND       P0004A	// L_2nd SUPPORT BW
LOAD      M04060	// 06_L_2nd ROT Y IDLE 1st
OR        F00099
AND LOAD
AND       P00055	// L_P&P UP (SENSOR)
AND       P00045	// L_2nd PRESS RIGHT UP
AND       P00047	// L_2nd PRESS LEFT UP
AND       M01232	// LF ¢¬¨­AI ¨úE¢Ò¡À ¨ú¨¡¢¥O
OUT       M0308C	// -

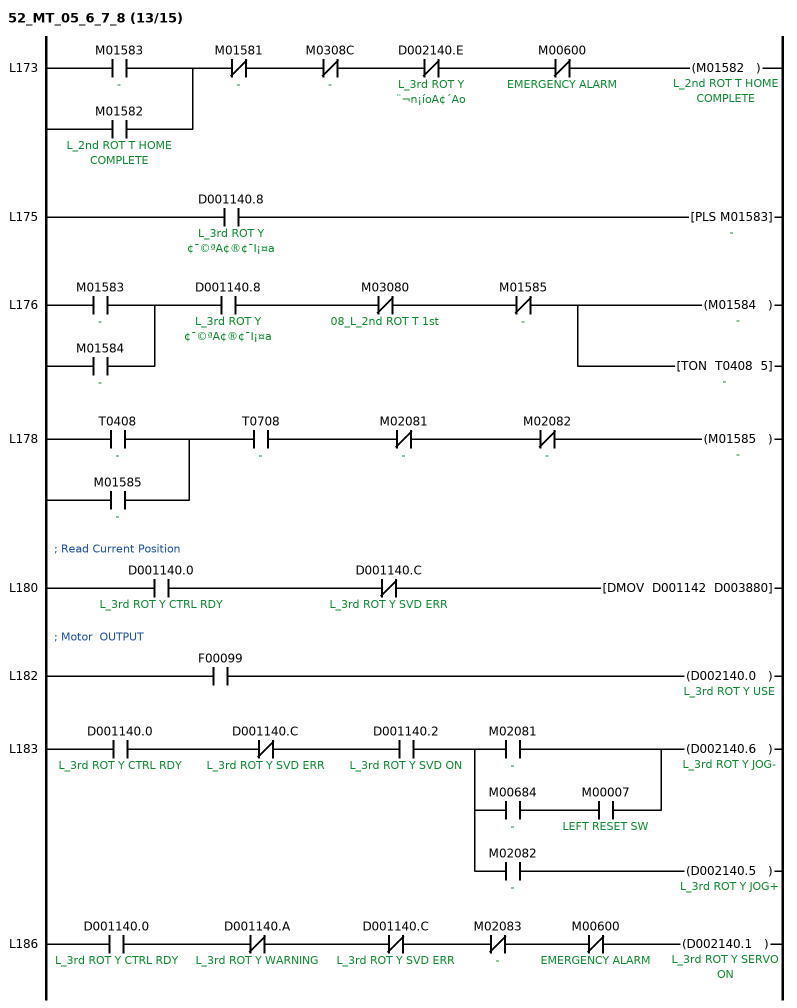
; L173
LOAD      M01583	// -
OR        M01582	// L_2nd ROT T HOME COMPLETE
AND NOT   M01581	// -
AND NOT   M0308C	// -
AND NOT   D002140.E	// L_3rd ROT Y ¨¬n¡íoA¢´Ao
AND NOT   M00600	// EMERGENCY ALARM
OUT       M01582	// L_2nd ROT T HOME COMPLETE
; L175
LOAD      D001140.8	// L_3rd ROT Y ¢¯©ªA¢®¢¯I¡¤a
OUTP      M01583	// -
; L176
LOAD      M01583	// -
OR        M01584	// -
AND       D001140.8	// L_3rd ROT Y ¢¯©ªA¢®¢¯I¡¤a
AND NOT   M03080	// 08_L_2nd ROT T 1st
AND NOT   M01585	// -
OUT       M01584	// -
TON       T0408 5	// -
; L178
LOAD      T0408	// -
OR        M01585	// -
AND       T0708	// -
AND NOT   M02081	// -
AND NOT   M02082	// -
OUT       M01585	// -
; L180
LOAD      D001140.0	// L_3rd ROT Y CTRL RDY
AND NOT   D001140.C	// L_3rd ROT Y SVD ERR
DMOV      D001142 D003880
// output comment: Read Current Position
//  Motor  OUTPUT
; L182
LOAD      F00099
OUT       D002140.0	// L_3rd ROT Y USE
; L183
LOAD      D001140.0	// L_3rd ROT Y CTRL RDY
AND NOT   D001140.C	// L_3rd ROT Y SVD ERR
AND       D001140.2	// L_3rd ROT Y SVD ON
MPUSH
LOAD      M02081	// -
LOAD      M00684	// -
AND       M00007	// LEFT RESET SW
OR LOAD
AND LOAD
OUT       D002140.6	// L_3rd ROT Y JOG-
MPOP
AND       M02082	// -
OUT       D002140.5	// L_3rd ROT Y JOG+
; L186
LOAD      D001140.0	// L_3rd ROT Y CTRL RDY
AND NOT   D001140.A	// L_3rd ROT Y WARNING
AND NOT   D001140.C	// L_3rd ROT Y SVD ERR
AND NOT   M02083	// -
AND NOT   M00600	// EMERGENCY ALARM
OUT       D002140.1	// L_3rd ROT Y SERVO ON

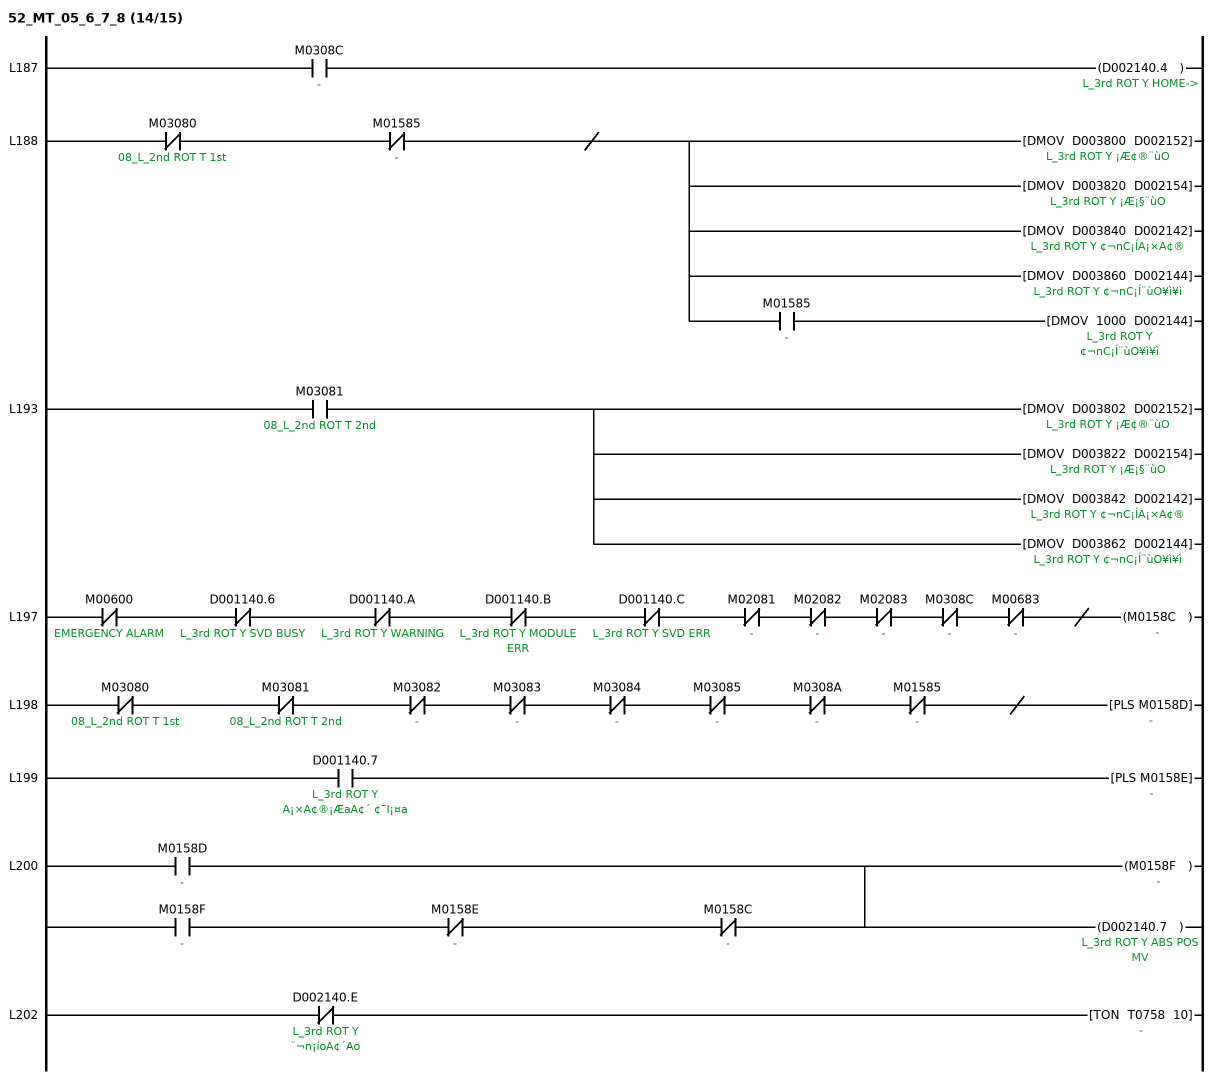
; L187
LOAD      M0308C	// -
OUT       D002140.4	// L_3rd ROT Y HOME->
; L188
LOAD NOT  M03080	// 08_L_2nd ROT T 1st
AND NOT   M01585	// -
NOT
DMOV      D003800 D002152	// L_3rd ROT Y ¡Æ¢®¨ùO
DMOV      D003820 D002154	// L_3rd ROT Y ¡Æ¡§¨ùO
DMOV      D003840 D002142	// L_3rd ROT Y ¢¬nC¡ÍA¡×A¢®
DMOV      D003860 D002144	// L_3rd ROT Y ¢¬nC¡Í¨ùO¥ì¥ì
AND       M01585	// -
DMOV      1000 D002144	// L_3rd ROT Y ¢¬nC¡Í¨ùO¥ì¥ì
; L193
LOAD      M03081	// 08_L_2nd ROT T 2nd
DMOV      D003802 D002152	// L_3rd ROT Y ¡Æ¢®¨ùO
DMOV      D003822 D002154	// L_3rd ROT Y ¡Æ¡§¨ùO
DMOV      D003842 D002142	// L_3rd ROT Y ¢¬nC¡ÍA¡×A¢®
DMOV      D003862 D002144	// L_3rd ROT Y ¢¬nC¡Í¨ùO¥ì¥ì
; L197
LOAD NOT  M00600	// EMERGENCY ALARM
AND NOT   D001140.6	// L_3rd ROT Y SVD BUSY
AND NOT   D001140.A	// L_3rd ROT Y WARNING
AND NOT   D001140.B	// L_3rd ROT Y MODULE ERR
AND NOT   D001140.C	// L_3rd ROT Y SVD ERR
AND NOT   M02081	// -
AND NOT   M02082	// -
AND NOT   M02083	// -
AND NOT   M0308C	// -
AND NOT   M00683	// -
NOT
OUT       M0158C	// -
; L198
LOAD NOT  M03080	// 08_L_2nd ROT T 1st
AND NOT   M03081	// 08_L_2nd ROT T 2nd
AND NOT   M03082	// -
AND NOT   M03083	// -
AND NOT   M03084	// -
AND NOT   M03085	// -
AND NOT   M0308A	// -
AND NOT   M01585	// -
NOT
OUTP      M0158D	// -
; L199
LOAD      D001140.7	// L_3rd ROT Y A¡×A¢®¡ÆaA¢´ ¢¯I¡¤a
OUTP      M0158E	// -
; L200
LOAD      M0158D	// -
LOAD      M0158F	// -
AND NOT   M0158E	// -
AND NOT   M0158C	// -
OR LOAD
OUT       M0158F	// -
OUT       D002140.7	// L_3rd ROT Y ABS POS MV
; L202
LOAD NOT  D002140.E	// L_3rd ROT Y ¨¬n¡íoA¢´Ao
TON       T0758 10	// -

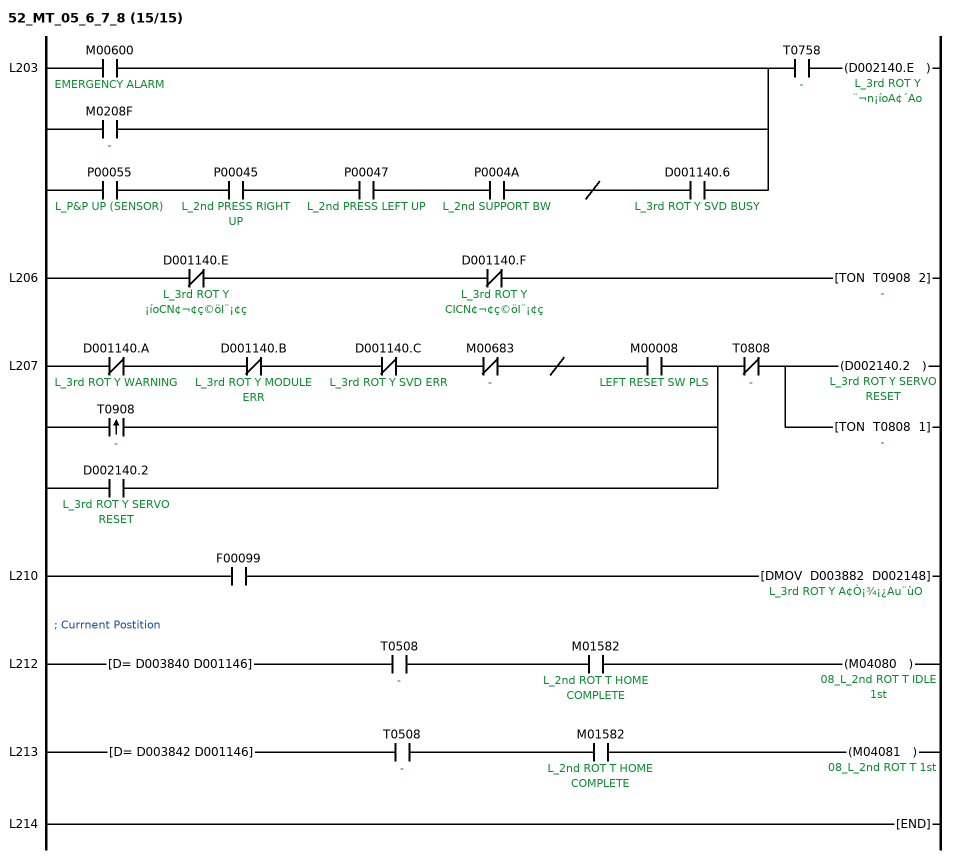
; L203
LOAD      M00600	// EMERGENCY ALARM
OR        M0208F	// -
LOAD      P00055	// L_P&P UP (SENSOR)
AND       P00045	// L_2nd PRESS RIGHT UP
AND       P00047	// L_2nd PRESS LEFT UP
AND       P0004A	// L_2nd SUPPORT BW
NOT
AND       D001140.6	// L_3rd ROT Y SVD BUSY
OR LOAD
AND       T0758	// -
OUT       D002140.E	// L_3rd ROT Y ¨¬n¡íoA¢´Ao
; L206
LOAD NOT  D001140.E	// L_3rd ROT Y ¡íoCN¢¬¢ç©öI¨¡¢ç
AND NOT   D001140.F	// L_3rd ROT Y CICN¢¬¢ç©öI¨¡¢ç
TON       T0908 2	// -
; L207
LOAD NOT  D001140.A	// L_3rd ROT Y WARNING
AND NOT   D001140.B	// L_3rd ROT Y MODULE ERR
AND NOT   D001140.C	// L_3rd ROT Y SVD ERR
AND NOT   M00683	// -
NOT
AND       M00008	// LEFT RESET SW PLS
ORP       T0908	// -
OR        D002140.2	// L_3rd ROT Y SERVO RESET
AND NOT   T0808	// -
OUT       D002140.2	// L_3rd ROT Y SERVO RESET
TON       T0808 1	// -
; L210
LOAD      F00099
DMOV      D003882 D002148	// L_3rd ROT Y A¢Ò¡¾¡¿Au¨ùO
// Currnent Postition
; L212
LOADD=    D003840 D001146
AND       T0508	// -
AND       M01582	// L_2nd ROT T HOME COMPLETE
OUT       M04080	// 08_L_2nd ROT T IDLE 1st
; L213
LOADD=    D003842 D001146
AND       T0508	// -
AND       M01582	// L_2nd ROT T HOME COMPLETE
OUT       M04081	// 08_L_2nd ROT T 1st
; L214
END

PROGRAM 53_MT_09_10_11_12 (task: ¨ö¨¬A¥ì CA¡¤I¡¾¡¿¡¤¡Í)

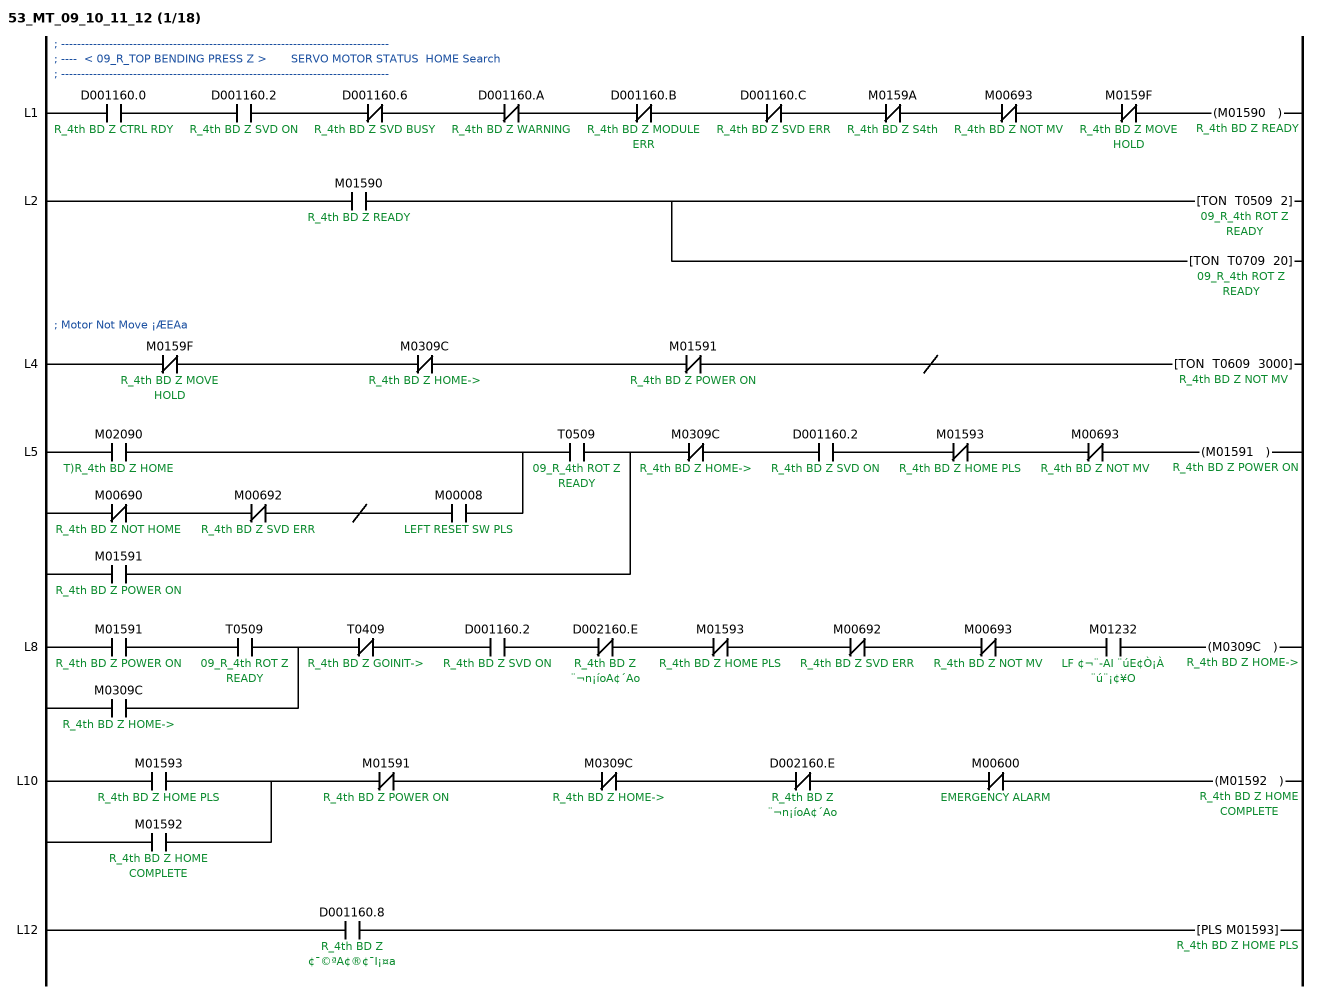
// ----------------------------------------------------------------------------------
// 
// ----  < 09_R_TOP BENDING PRESS Z >       SERVO MOTOR STATUS  HOME Search
// 
// ----------------------------------------------------------------------------------
; L1
LOAD      D001160.0	// R_4th BD Z CTRL RDY
AND       D001160.2	// R_4th BD Z SVD ON
AND NOT   D001160.6	// R_4th BD Z SVD BUSY
AND NOT   D001160.A	// R_4th BD Z WARNING
AND NOT   D001160.B	// R_4th BD Z MODULE ERR
AND NOT   D001160.C	// R_4th BD Z SVD ERR
AND NOT   M0159A	// R_4th BD Z S4th
AND NOT   M00693	// R_4th BD Z NOT MV
AND NOT   M0159F	// R_4th BD Z MOVE HOLD
OUT       M01590	// R_4th BD Z READY
; L2
LOAD      M01590	// R_4th BD Z READY
TON       T0509 2	// 09_R_4th ROT Z READY
TON       T0709 20	// 09_R_4th ROT Z READY
; L4
LOAD NOT  M0159F	// R_4th BD Z MOVE HOLD
AND NOT   M0309C	// R_4th BD Z HOME->
AND NOT   M01591	// R_4th BD Z POWER ON
NOT
TON       T0609 3000	// R_4th BD Z NOT MV
// output comment: Motor Not Move ¡ÆEAa
; L5
LOAD      M02090	// T)R_4th BD Z HOME
LOAD NOT  M00690	// R_4th BD Z NOT HOME
AND NOT   M00692	// R_4th BD Z SVD ERR
NOT
AND       M00008	// LEFT RESET SW PLS
OR LOAD
AND       T0509	// 09_R_4th ROT Z READY
OR        M01591	// R_4th BD Z POWER ON
AND NOT   M0309C	// R_4th BD Z HOME->
AND       D001160.2	// R_4th BD Z SVD ON
AND NOT   M01593	// R_4th BD Z HOME PLS
AND NOT   M00693	// R_4th BD Z NOT MV
OUT       M01591	// R_4th BD Z POWER ON
; L8
LOAD      M01591	// R_4th BD Z POWER ON
AND       T0509	// 09_R_4th ROT Z READY
OR        M0309C	// R_4th BD Z HOME->
AND NOT   T0409	// R_4th BD Z GOINIT->
AND       D001160.2	// R_4th BD Z SVD ON
AND NOT   D002160.E	// R_4th BD Z ¨¬n¡íoA¢´Ao
AND NOT   M01593	// R_4th BD Z HOME PLS
AND NOT   M00692	// R_4th BD Z SVD ERR
AND NOT   M00693	// R_4th BD Z NOT MV
AND       M01232	// LF ¢¬¨­AI ¨úE¢Ò¡À ¨ú¨¡¢¥O
OUT       M0309C	// R_4th BD Z HOME->
; L10
LOAD      M01593	// R_4th BD Z HOME PLS
OR        M01592	// R_4th BD Z HOME COMPLETE
AND NOT   M01591	// R_4th BD Z POWER ON
AND NOT   M0309C	// R_4th BD Z HOME->
AND NOT   D002160.E	// R_4th BD Z ¨¬n¡íoA¢´Ao
AND NOT   M00600	// EMERGENCY ALARM
OUT       M01592	// R_4th BD Z HOME COMPLETE
; L12
LOAD      D001160.8	// R_4th BD Z ¢¯©ªA¢®¢¯I¡¤a
OUTP      M01593	// R_4th BD Z HOME PLS

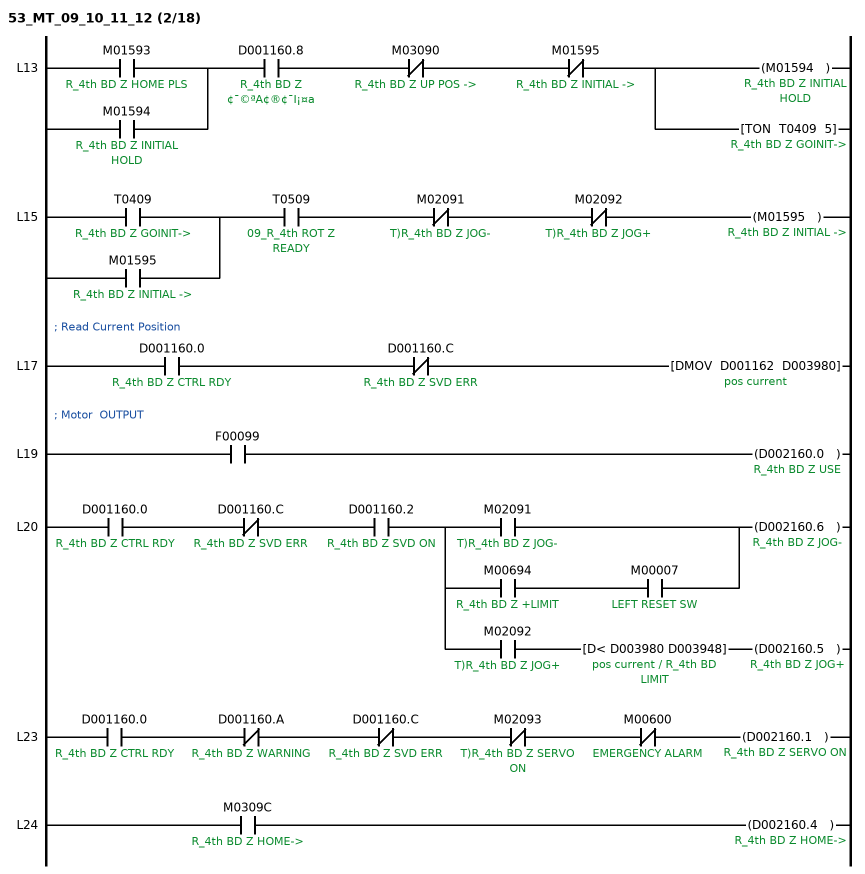
; L13
LOAD      M01593	// R_4th BD Z HOME PLS
OR        M01594	// R_4th BD Z INITIAL HOLD
AND       D001160.8	// R_4th BD Z ¢¯©ªA¢®¢¯I¡¤a
AND NOT   M03090	// R_4th BD Z UP POS ->
AND NOT   M01595	// R_4th BD Z INITIAL ->
OUT       M01594	// R_4th BD Z INITIAL HOLD
TON       T0409 5	// R_4th BD Z GOINIT->
; L15
LOAD      T0409	// R_4th BD Z GOINIT->
OR        M01595	// R_4th BD Z INITIAL ->
AND       T0509	// 09_R_4th ROT Z READY
AND NOT   M02091	// T)R_4th BD Z JOG-
AND NOT   M02092	// T)R_4th BD Z JOG+
OUT       M01595	// R_4th BD Z INITIAL ->
; L17
LOAD      D001160.0	// R_4th BD Z CTRL RDY
AND NOT   D001160.C	// R_4th BD Z SVD ERR
DMOV      D001162 D003980	// pos current
// output comment: Read Current Position
//  Motor  OUTPUT
; L19
LOAD      F00099
OUT       D002160.0	// R_4th BD Z USE
; L20
LOAD      D001160.0	// R_4th BD Z CTRL RDY
AND NOT   D001160.C	// R_4th BD Z SVD ERR
AND       D001160.2	// R_4th BD Z SVD ON
MPUSH
LOAD      M02091	// T)R_4th BD Z JOG-
LOAD      M00694	// R_4th BD Z +LIMIT
AND       M00007	// LEFT RESET SW
OR LOAD
AND LOAD
OUT       D002160.6	// R_4th BD Z JOG-
MPOP
AND       M02092	// T)R_4th BD Z JOG+
ANDD<     D003980 D003948	// pos current / R_4th BD LIMIT
OUT       D002160.5	// R_4th BD Z JOG+
; L23
LOAD      D001160.0	// R_4th BD Z CTRL RDY
AND NOT   D001160.A	// R_4th BD Z WARNING
AND NOT   D001160.C	// R_4th BD Z SVD ERR
AND NOT   M02093	// T)R_4th BD Z SERVO ON
AND NOT   M00600	// EMERGENCY ALARM
OUT       D002160.1	// R_4th BD Z SERVO ON
; L24
LOAD      M0309C	// R_4th BD Z HOME->
OUT       D002160.4	// R_4th BD Z HOME->

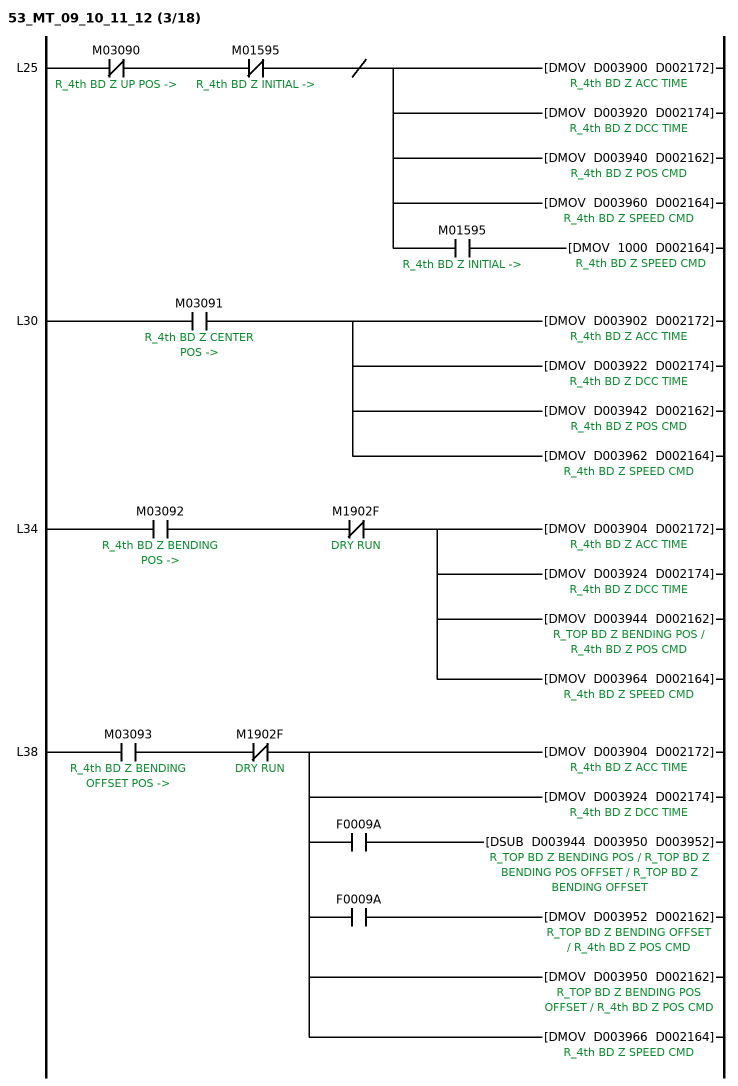
; L25
LOAD NOT  M03090	// R_4th BD Z UP POS ->
AND NOT   M01595	// R_4th BD Z INITIAL ->
NOT
DMOV      D003900 D002172	// R_4th BD Z ACC TIME
DMOV      D003920 D002174	// R_4th BD Z DCC TIME
DMOV      D003940 D002162	// R_4th BD Z POS CMD
DMOV      D003960 D002164	// R_4th BD Z SPEED CMD
AND       M01595	// R_4th BD Z INITIAL ->
DMOV      1000 D002164	// R_4th BD Z SPEED CMD
; L30
LOAD      M03091	// R_4th BD Z CENTER POS ->
DMOV      D003902 D002172	// R_4th BD Z ACC TIME
DMOV      D003922 D002174	// R_4th BD Z DCC TIME
DMOV      D003942 D002162	// R_4th BD Z POS CMD
DMOV      D003962 D002164	// R_4th BD Z SPEED CMD
; L34
LOAD      M03092	// R_4th BD Z BENDING POS ->
AND NOT   M1902F	// DRY RUN
DMOV      D003904 D002172	// R_4th BD Z ACC TIME
DMOV      D003924 D002174	// R_4th BD Z DCC TIME
DMOV      D003944 D002162	// R_TOP BD Z BENDING POS / R_4th BD Z POS CMD
DMOV      D003964 D002164	// R_4th BD Z SPEED CMD
; L38
LOAD      M03093	// R_4th BD Z BENDING OFFSET POS ->
AND NOT   M1902F	// DRY RUN
DMOV      D003904 D002172	// R_4th BD Z ACC TIME
DMOV      D003924 D002174	// R_4th BD Z DCC TIME
MPUSH
AND       F0009A
DSUB      D003944 D003950 D003952	// R_TOP BD Z BENDING POS / R_TOP BD Z BENDING POS OFFSET / R_TOP BD Z BENDING OFFSET
MLOAD
AND       F0009A
DMOV      D003952 D002162	// R_TOP BD Z BENDING OFFSET / R_4th BD Z POS CMD
MPOP
DMOV      D003950 D002162	// R_TOP BD Z BENDING POS OFFSET / R_4th BD Z POS CMD
DMOV      D003966 D002164	// R_4th BD Z SPEED CMD

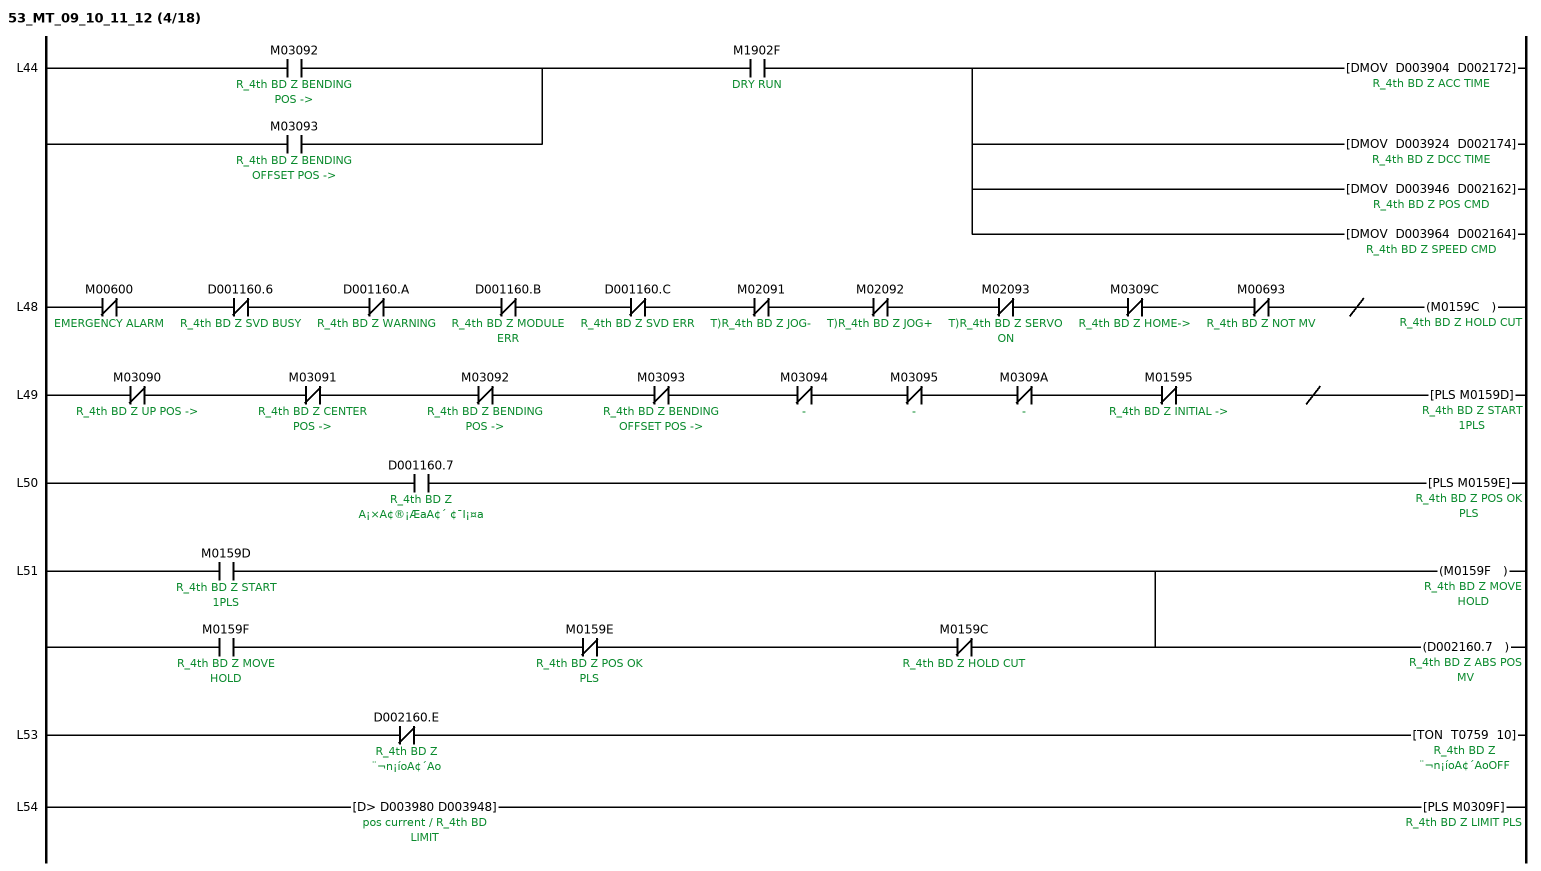
; L44
LOAD      M03092	// R_4th BD Z BENDING POS ->
OR        M03093	// R_4th BD Z BENDING OFFSET POS ->
AND       M1902F	// DRY RUN
DMOV      D003904 D002172	// R_4th BD Z ACC TIME
DMOV      D003924 D002174	// R_4th BD Z DCC TIME
DMOV      D003946 D002162	// R_4th BD Z POS CMD
DMOV      D003964 D002164	// R_4th BD Z SPEED CMD
; L48
LOAD NOT  M00600	// EMERGENCY ALARM
AND NOT   D001160.6	// R_4th BD Z SVD BUSY
AND NOT   D001160.A	// R_4th BD Z WARNING
AND NOT   D001160.B	// R_4th BD Z MODULE ERR
AND NOT   D001160.C	// R_4th BD Z SVD ERR
AND NOT   M02091	// T)R_4th BD Z JOG-
AND NOT   M02092	// T)R_4th BD Z JOG+
AND NOT   M02093	// T)R_4th BD Z SERVO ON
AND NOT   M0309C	// R_4th BD Z HOME->
AND NOT   M00693	// R_4th BD Z NOT MV
NOT
OUT       M0159C	// R_4th BD Z HOLD CUT
; L49
LOAD NOT  M03090	// R_4th BD Z UP POS ->
AND NOT   M03091	// R_4th BD Z CENTER POS ->
AND NOT   M03092	// R_4th BD Z BENDING POS ->
AND NOT   M03093	// R_4th BD Z BENDING OFFSET POS ->
AND NOT   M03094	// -
AND NOT   M03095	// -
AND NOT   M0309A	// -
AND NOT   M01595	// R_4th BD Z INITIAL ->
NOT
OUTP      M0159D	// R_4th BD Z START 1PLS
; L50
LOAD      D001160.7	// R_4th BD Z A¡×A¢®¡ÆaA¢´ ¢¯I¡¤a
OUTP      M0159E	// R_4th BD Z POS OK PLS
; L51
LOAD      M0159D	// R_4th BD Z START 1PLS
LOAD      M0159F	// R_4th BD Z MOVE HOLD
AND NOT   M0159E	// R_4th BD Z POS OK PLS
AND NOT   M0159C	// R_4th BD Z HOLD CUT
OR LOAD
OUT       M0159F	// R_4th BD Z MOVE HOLD
OUT       D002160.7	// R_4th BD Z ABS POS MV
; L53
LOAD NOT  D002160.E	// R_4th BD Z ¨¬n¡íoA¢´Ao
TON       T0759 10	// R_4th BD Z ¨¬n¡íoA¢´AoOFF
; L54
LOADD>    D003980 D003948	// pos current / R_4th BD LIMIT
OUTP      M0309F	// R_4th BD Z LIMIT PLS

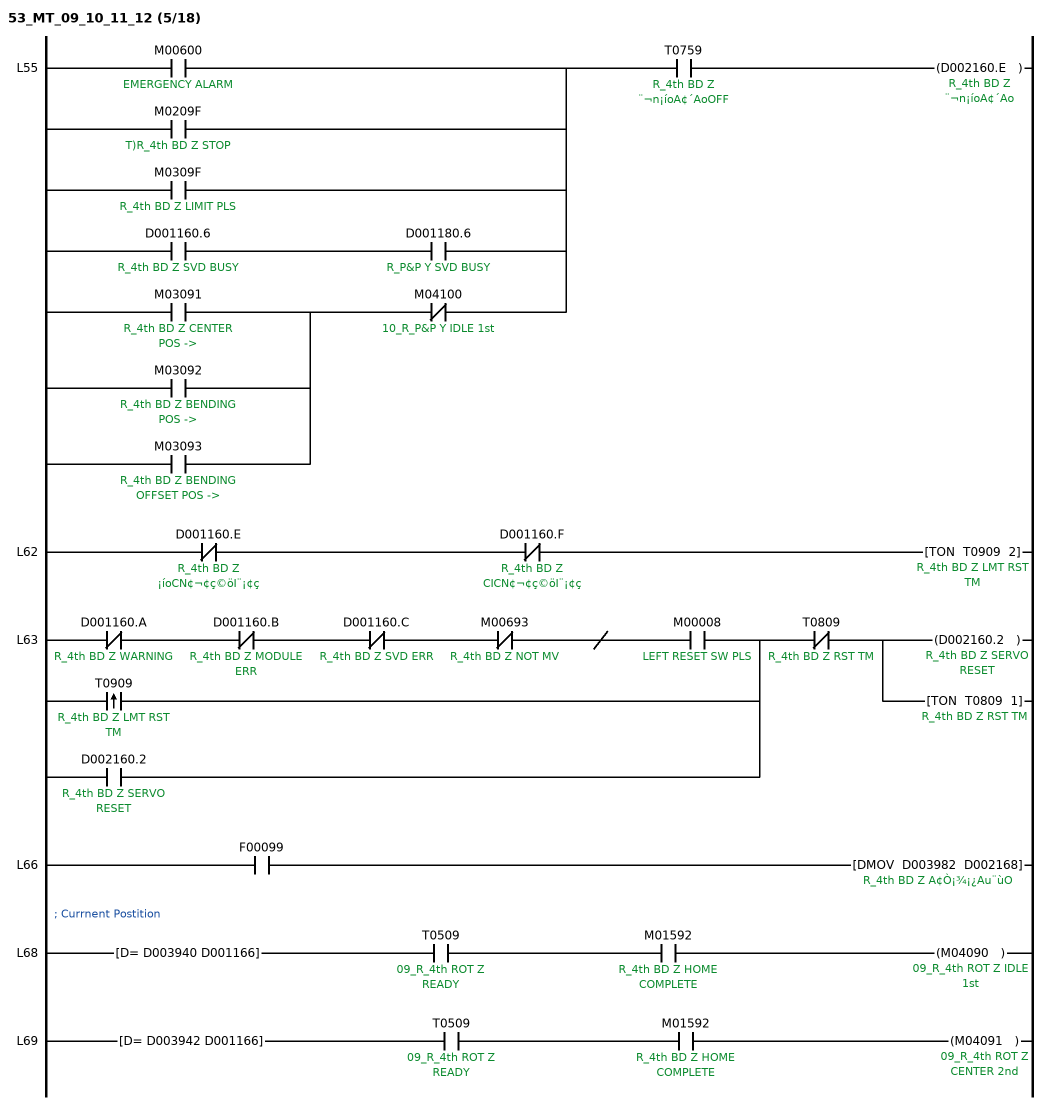
; L55
LOAD      M00600	// EMERGENCY ALARM
OR        M0209F	// T)R_4th BD Z STOP
OR        M0309F	// R_4th BD Z LIMIT PLS
LOAD      D001160.6	// R_4th BD Z SVD BUSY
AND       D001180.6	// R_P&P Y SVD BUSY
OR LOAD
LOAD      M03091	// R_4th BD Z CENTER POS ->
OR        M03092	// R_4th BD Z BENDING POS ->
OR        M03093	// R_4th BD Z BENDING OFFSET POS ->
AND NOT   M04100	// 10_R_P&P Y IDLE 1st
OR LOAD
AND       T0759	// R_4th BD Z ¨¬n¡íoA¢´AoOFF
OUT       D002160.E	// R_4th BD Z ¨¬n¡íoA¢´Ao
; L62
LOAD NOT  D001160.E	// R_4th BD Z ¡íoCN¢¬¢ç©öI¨¡¢ç
AND NOT   D001160.F	// R_4th BD Z CICN¢¬¢ç©öI¨¡¢ç
TON       T0909 2	// R_4th BD Z LMT RST TM
; L63
LOAD NOT  D001160.A	// R_4th BD Z WARNING
AND NOT   D001160.B	// R_4th BD Z MODULE ERR
AND NOT   D001160.C	// R_4th BD Z SVD ERR
AND NOT   M00693	// R_4th BD Z NOT MV
NOT
AND       M00008	// LEFT RESET SW PLS
ORP       T0909	// R_4th BD Z LMT RST TM
OR        D002160.2	// R_4th BD Z SERVO RESET
AND NOT   T0809	// R_4th BD Z RST TM
OUT       D002160.2	// R_4th BD Z SERVO RESET
TON       T0809 1	// R_4th BD Z RST TM
; L66
LOAD      F00099
DMOV      D003982 D002168	// R_4th BD Z A¢Ò¡¾¡¿Au¨ùO
// Currnent Postition
; L68
LOADD=    D003940 D001166
AND       T0509	// 09_R_4th ROT Z READY
AND       M01592	// R_4th BD Z HOME COMPLETE
OUT       M04090	// 09_R_4th ROT Z IDLE 1st
; L69
LOADD=    D003942 D001166
AND       T0509	// 09_R_4th ROT Z READY
AND       M01592	// R_4th BD Z HOME COMPLETE
OUT       M04091	// 09_R_4th ROT Z CENTER 2nd

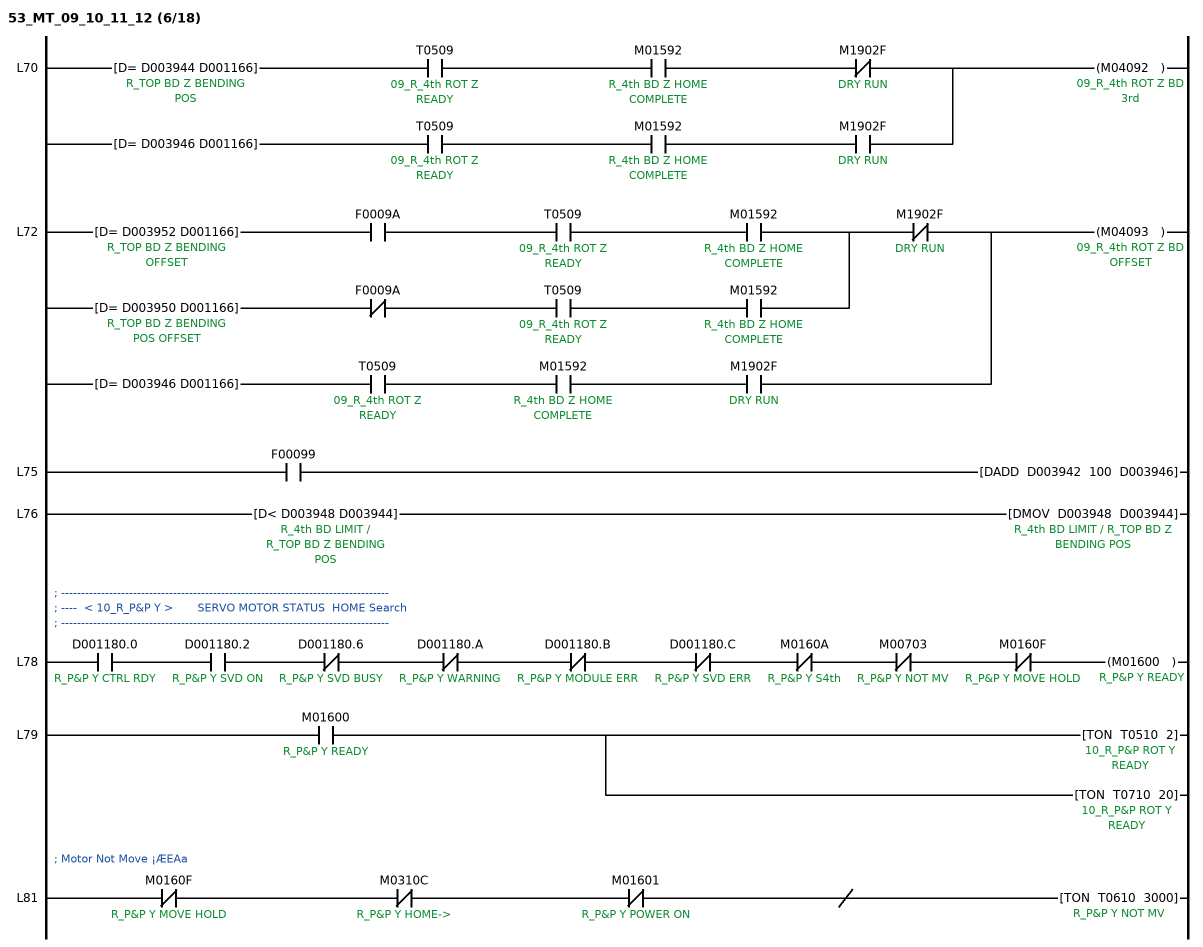
; L70
LOADD=    D003944 D001166	// R_TOP BD Z BENDING POS
AND       T0509	// 09_R_4th ROT Z READY
AND       M01592	// R_4th BD Z HOME COMPLETE
AND NOT   M1902F	// DRY RUN
LOADD=    D003946 D001166
AND       T0509	// 09_R_4th ROT Z READY
AND       M01592	// R_4th BD Z HOME COMPLETE
AND       M1902F	// DRY RUN
OR LOAD
OUT       M04092	// 09_R_4th ROT Z BD 3rd
; L72
LOADD=    D003952 D001166	// R_TOP BD Z BENDING OFFSET
AND       F0009A
AND       T0509	// 09_R_4th ROT Z READY
AND       M01592	// R_4th BD Z HOME COMPLETE
LOADD=    D003950 D001166	// R_TOP BD Z BENDING POS OFFSET
AND NOT   F0009A
AND       T0509	// 09_R_4th ROT Z READY
AND       M01592	// R_4th BD Z HOME COMPLETE
OR LOAD
AND NOT   M1902F	// DRY RUN
LOADD=    D003946 D001166
AND       T0509	// 09_R_4th ROT Z READY
AND       M01592	// R_4th BD Z HOME COMPLETE
AND       M1902F	// DRY RUN
OR LOAD
OUT       M04093	// 09_R_4th ROT Z BD OFFSET
; L75
LOAD      F00099
DADD      D003942 100 D003946
; L76
LOADD<    D003948 D003944	// R_4th BD LIMIT / R_TOP BD Z BENDING POS
DMOV      D003948 D003944	// R_4th BD LIMIT / R_TOP BD Z BENDING POS
// ----------------------------------------------------------------------------------
// 
// ----  < 10_R_P&P Y >       SERVO MOTOR STATUS  HOME Search
// 
// ----------------------------------------------------------------------------------
; L78
LOAD      D001180.0	// R_P&P Y CTRL RDY
AND       D001180.2	// R_P&P Y SVD ON
AND NOT   D001180.6	// R_P&P Y SVD BUSY
AND NOT   D001180.A	// R_P&P Y WARNING
AND NOT   D001180.B	// R_P&P Y MODULE ERR
AND NOT   D001180.C	// R_P&P Y SVD ERR
AND NOT   M0160A	// R_P&P Y S4th
AND NOT   M00703	// R_P&P Y NOT MV
AND NOT   M0160F	// R_P&P Y MOVE HOLD
OUT       M01600	// R_P&P Y READY
; L79
LOAD      M01600	// R_P&P Y READY
TON       T0510 2	// 10_R_P&P ROT Y READY
TON       T0710 20	// 10_R_P&P ROT Y READY
; L81
LOAD NOT  M0160F	// R_P&P Y MOVE HOLD
AND NOT   M0310C	// R_P&P Y HOME->
AND NOT   M01601	// R_P&P Y POWER ON
NOT
TON       T0610 3000	// R_P&P Y NOT MV
// output comment: Motor Not Move ¡ÆEAa

